C03641=1047.651,269.816,394.921,172.009,38.848,157.370
C03642=1047.658,270.065,394.890,172.012,38.851,157.371
C03643=1047.664,270.312,394.860,172.016,38.854,157.372
C03644=1047.670,270.561,394.829,172.018,38.856,157.372
C03645=1047.677,270.809,394.799,172.021,38.859,157.373
C03646=1047.683,271.057,394.769,172.023,38.862,157.374
C03647=1047.690,271.305,394.738,172.027,38.865,157.375
C03648=1047.697,271.553,394.708,172.030,38.868,157.375
C03649=1047.703,271.801,394.678,172.032,38.871,157.376
C03650=1047.710,272.049,394.648,172.036,38.874,157.377
C03651=1047.717,272.297,394.616,172.039,38.876,157.377
C03652=1047.723,272.545,394.586,172.041,38.879,157.378
C03653=1047.730,272.793,394.556,172.045,38.882,157.379
C03654=1047.736,273.041,394.525,172.047,38.885,157.379
C03655=1047.742,273.290,394.495,172.050,38.888,157.380
C03656=1047.749,273.537,394.464,172.054,38.891,157.381
C03657=1047.755,273.785,394.433,172.056,38.893,157.381
C03658=1047.762,274.034,394.403,172.059,38.896,157.382
C03659=1047.769,274.282,394.373,172.063,38.899,157.383
C03660=1047.775,274.529,394.342,172.065,38.902,157.384
C03661=1047.781,274.778,394.311,172.068,38.905,157.384
C03662=1047.789,275.026,394.281,172.072,38.908,157.385
C03663=1047.795,275.274,394.249,172.074,38.910,157.386
C03664=1047.801,275.521,394.219,172.077,38.913,157.386
C03665=1047.807,275.770,394.188,172.081,38.917,157.387
C03666=1047.815,276.018,394.157,172.083,38.919,157.388
C03667=1047.821,276.265,394.127,172.087,38.922,157.389
C03668=1047.828,276.535,394.093,172.089,38.925,157.389
C03669=1047.835,276.805,394.060,172.093,38.929,157.390
C03670=1047.842,277.075,394.026,172.096,38.931,157.391
C03671=1047.850,277.344,393.993,172.100,38.935,157.392
C03672=1047.856,277.592,393.962,172.102,38.938,157.392
C03673=1047.863,277.840,393.931,172.106,38.940,157.393
C03674=1047.869,278.089,393.900,172.109,38.943,157.394
C03675=1047.877,278.336,393.869,172.112,38.946,157.394
C03676=1047.882,278.584,393.839,172.115,38.949,157.395
C03677=1047.889,278.832,393.807,172.118,38.952,157.396
C03678=1047.895,279.081,393.777,172.121,38.955,157.397
C03679=1047.902,279.329,393.745,172.124,38.958,157.397
C03680=1047.908,279.576,393.714,172.128,38.961,157.398
C03681=1047.915,279.824,393.684,172.130,38.964,157.399
C03682=1047.921,280.072,393.652,172.133,38.966,157.399
C03683=1047.928,280.320,393.621,172.137,38.970,157.400
C03684=1047.935,280.569,393.590,172.139,38.973,157.401
C03685=1047.941,280.816,393.559,172.143,38.975,157.402
C03686=1047.947,281.064,393.527,172.145,38.978,157.402
C03687=1047.954,281.312,393.497,172.148,38.982,157.403
C03688=1047.961,281.560,393.465,172.152,38.984,157.404
C03689=1047.967,281.808,393.434,172.155,38.987,157.405
C03690=1047.973,282.055,393.403,172.158,38.990,157.405
C03691=1047.980,282.304,393.372,172.161,38.993,157.406
C03692=1047.987,282.552,393.341,172.165,38.996,157.407
C03693=1047.993,282.800,393.309,172.167,38.999,157.408
C03694=1048.000,283.048,393.278,172.171,39.002,157.408
C03695=1048.007,283.295,393.246,172.174,39.005,157.409
C03696=1048.013,283.544,393.216,172.177,39.008,157.410
C03697=1048.020,283.792,393.184,172.180,39.011,157.411
C03698=1048.026,284.039,393.153,172.184,39.014,157.411
C03699=1048.033,284.287,393.122,172.186,39.017,157.412
C03700=1048.040,284.535,393.090,172.189,39.020,157.413
C03701=1048.046,284.783,393.059,172.193,39.023,157.413
C03702=1048.053,285.031,393.027,172.195,39.026,157.414
C03703=1048.060,285.279,392.996,172.199,39.028,157.415
C03704=1048.066,285.526,392.965,172.202,39.032,157.416
C03705=1048.073,285.774,392.933,172.205,39.035,157.416
C03706=1048.080,286.022,392.902,172.209,39.037,157.417
C03707=1048.087,286.270,392.870,172.212,39.040,157.418
C03708=1048.093,286.518,392.839,172.216,39.044,157.419
C03709=1048.100,286.766,392.807,172.218,39.046,157.419
C03710=1048.106,287.014,392.775,172.222,39.049,157.420
C03711=1048.113,287.262,392.744,172.224,39.052,157.421
C03712=1048.119,287.510,392.713,172.228,39.055,157.422
C03713=1048.126,287.758,392.681,172.231,39.058,157.422
C03714=1048.133,288.006,392.650,172.235,39.061,157.423
C03715=1048.140,288.254,392.618,172.237,39.064,157.424
C03716=1048.146,288.502,392.586,172.241,39.067,157.425
C03717=1048.152,288.750,392.555,172.244,39.070,157.425
C03718=1048.159,288.997,392.523,172.247,39.073,157.426
C03719=1048.166,289.245,392.491,172.250,39.076,157.427
C03720=1048.172,289.493,392.459,172.254,39.079,157.428
C03721=1048.179,289.741,392.428,172.258,39.082,157.428
C03722=1048.186,289.989,392.396,172.260,39.085,157.429
C03723=1048.193,290.236,392.364,172.264,39.088,157.430
C03724=1048.200,290.518,392.328,172.268,39.092,157.431
C03725=1048.207,290.799,392.292,172.271,39.095,157.432
C03726=1048.215,291.080,392.255,172.274,39.099,157.433
C03727=1048.222,291.361,392.219,172.278,39.102,157.433
C03728=1048.229,291.610,392.187,172.282,39.105,157.434
C03729=1048.236,291.857,392.156,172.285,39.108,157.435
C03730=1048.242,292.105,392.123,172.288,39.111,157.436
C03731=1048.249,292.353,392.092,172.292,39.114,157.436
C03732=1048.255,292.601,392.060,172.295,39.118,157.437
C03733=1048.262,292.848,392.027,172.298,39.120,157.438
C03734=1048.268,293.096,391.996,172.301,39.123,157.439
C03735=1048.275,293.344,391.964,172.305,39.127,157.440
C03736=1048.281,293.592,391.932,172.309,39.129,157.440
C03737=1048.288,293.839,391.900,172.311,39.133,157.441
C03738=1048.295,294.088,391.867,172.315,39.135,157.442
C03739=1048.302,294.335,391.835,172.319,39.139,157.443
C03740=1048.308,294.584,391.803,172.321,39.142,157.443
C03741=1048.315,294.831,391.771,172.325,39.145,157.444
C03742=1048.322,295.079,391.740,172.328,39.148,157.445
C03743=1048.328,295.326,391.707,172.332,39.151,157.446
C03744=1048.335,295.574,391.675,172.335,39.154,157.447
C03745=1048.342,295.823,391.642,172.338,39.157,157.447
C03746=1048.349,296.070,391.610,172.342,39.160,157.448
C03747=1048.355,296.317,391.577,172.346,39.163,157.449
C03748=1048.361,296.566,391.545,172.348,39.167,157.450
C03749=1048.367,296.813,391.513,172.352,39.170,157.450
C03750=1048.374,297.061,391.480,172.356,39.173,157.451
C03751=1048.381,297.308,391.448,172.359,39.176,157.452
C03752=1048.387,297.557,391.415,172.363,39.180,157.453
C03753=1048.393,297.805,391.383,172.365,39.182,157.454
C03754=1048.400,298.052,391.350,172.369,39.186,157.455
C03755=1048.406,298.300,391.317,172.373,39.189,157.455
C03756=1048.413,298.547,391.285,172.375,39.192,157.456
C03757=1048.419,298.795,391.252,172.379,39.195,157.457
C03758=1048.426,299.043,391.219,172.383,39.199,157.458
C03759=1048.432,299.291,391.187,172.386,39.202,157.459
C03760=1048.439,299.538,391.155,172.390,39.205,157.459
C03761=1048.446,299.786,391.122,172.393,39.208,157.460
C03762=1048.452,300.034,391.089,172.396,39.211,157.461
C03763=1048.459,300.282,391.056,172.400,39.214,157.462
C03764=1048.465,300.529,391.024,172.404,39.217,157.463
C03765=1048.471,300.777,390.991,172.407,39.221,157.464
C03766=1048.479,301.025,390.958,172.410,39.224,157.464
C03767=1048.485,301.273,390.926,172.414,39.227,157.465
C03768=1048.492,301.520,390.893,172.418,39.230,157.466
C03769=1048.498,301.768,390.860,172.421,39.234,157.467
C03770=1048.505,302.016,390.827,172.424,39.237,157.468
C03771=1048.511,302.264,390.794,172.428,39.240,157.469
C03772=1048.518,302.511,390.762,172.432,39.243,157.469
C03773=1048.525,302.759,390.728,172.435,39.246,157.470
C03774=1048.532,303.006,390.696,172.438,39.250,157.471
C03775=1048.538,303.254,390.663,172.442,39.253,157.472
C03776=1048.545,303.502,390.630,172.446,39.256,157.473
C03777=1048.551,303.750,390.597,172.449,39.259,157.473
C03778=1048.558,303.997,390.565,172.453,39.263,157.474
C03779=1048.565,304.245,390.531,172.456,39.266,157.475
C03780=1048.573,304.542,390.491,172.460,39.270,157.476
C03781=1048.581,304.840,390.452,172.465,39.274,157.477
C03782=1048.589,305.137,390.412,172.469,39.278,157.478
C03783=1048.597,305.435,390.373,172.473,39.281,157.479
C03784=1048.604,305.682,390.340,172.477,39.285,157.480
C03785=1048.611,305.930,390.307,172.481,39.288,157.481
C03786=1048.617,306.178,390.274,172.484,39.291,157.482
C03787=1048.624,306.425,390.240,172.487,39.294,157.482
C03788=1048.630,306.673,390.207,172.491,39.297,157.483
C03789=1048.638,306.920,390.175,172.495,39.301,157.484
C03790=1048.645,307.168,390.141,172.499,39.304,157.485
C03791=1048.651,307.415,390.109,172.503,39.307,157.486
C03792=1048.658,307.664,390.075,172.506,39.311,157.487
C03793=1048.665,307.911,390.042,172.509,39.314,157.487
C03794=1048.671,308.159,390.009,172.513,39.317,157.488
C03795=1048.679,308.407,389.975,172.517,39.320,157.489
C03796=1048.685,308.654,389.942,172.521,39.323,157.490
C03797=1048.692,308.902,389.909,172.524,39.327,157.491
C03798=1048.699,309.149,389.876,172.528,39.330,157.492
C03799=1048.706,309.397,389.843,172.532,39.333,157.493
C03800=1048.713,309.644,389.810,172.535,39.337,157.493
C03801=1048.720,309.892,389.776,172.539,39.340,157.494
C03802=1048.726,310.140,389.743,172.542,39.343,157.495
C03803=1048.733,310.387,389.709,172.546,39.347,157.496
C03804=1048.740,310.636,389.676,172.550,39.350,157.497
C03805=1048.747,310.883,389.643,172.554,39.353,157.498
C03806=1048.754,311.130,389.609,172.558,39.356,157.498
C03807=1048.761,311.379,389.576,172.561,39.359,157.499
C03808=1048.768,311.626,389.542,172.565,39.363,157.500
C03809=1048.775,311.873,389.509,172.568,39.366,157.501
C03810=1048.782,312.122,389.476,172.572,39.369,157.502
C03811=1048.788,312.369,389.442,172.576,39.373,157.503
C03812=1048.796,312.616,389.409,172.580,39.376,157.504
C03813=1048.803,312.864,389.376,172.583,39.379,157.505
C03814=1048.809,313.111,389.342,172.587,39.383,157.506
C03815=1048.816,313.359,389.308,172.591,39.386,157.506
C03816=1048.822,313.606,389.274,172.595,39.390,157.507
C03817=1048.829,313.854,389.240,172.599,39.393,157.508
C03818=1048.836,314.102,389.206,172.603,39.397,157.509
C03819=1048.842,314.349,389.172,172.606,39.400,157.510
C03820=1048.849,314.597,389.138,172.610,39.403,157.511
C03821=1048.855,314.844,389.104,172.613,39.407,157.512
C03822=1048.862,315.092,389.070,172.617,39.411,157.513
C03823=1048.869,315.340,389.036,172.621,39.414,157.514
C03824=1048.875,315.587,389.002,172.625,39.417,157.514
C03825=1048.882,315.835,388.968,172.629,39.421,157.515
C03826=1048.888,316.083,388.934,172.633,39.424,157.516
C03827=1048.895,316.330,388.900,172.637,39.428,157.517
C03828=1048.902,316.578,388.866,172.641,39.432,157.518
C03829=1048.909,316.825,388.832,172.644,39.435,157.519
C03830=1048.915,317.073,388.798,172.648,39.438,157.520
C03831=1048.922,317.320,388.763,172.652,39.442,157.521
C03832=1048.929,317.568,388.729,172.655,39.445,157.522
C03833=1048.936,317.815,388.695,172.659,39.449,157.523
C03834=1048.942,318.063,388.661,172.663,39.452,157.524
C03835=1048.949,318.310,388.627,172.667,39.456,157.525
C03836=1048.957,318.612,388.586,172.672,39.460,157.526
C03837=1048.966,318.914,388.544,172.677,39.465,157.527
C03838=1048.974,319.216,388.502,172.681,39.469,157.528
C03839=1048.982,319.518,388.460,172.686,39.473,157.529
C03840=1048.989,319.765,388.425,172.690,39.477,157.530
C03841=1048.995,320.013,388.391,172.694,39.480,157.531
C03842=1049.002,320.260,388.357,172.698,39.484,157.532
C03843=1049.009,320.508,388.322,172.702,39.487,157.533
C03844=1049.016,320.755,388.288,172.706,39.491,157.534
C03845=1049.023,321.003,388.254,172.710,39.494,157.535
C03846=1049.030,321.250,388.219,172.714,39.498,157.536
C03847=1049.037,321.498,388.185,172.717,39.501,157.537
C03848=1049.043,321.746,388.150,172.721,39.505,157.538
C03849=1049.051,321.993,388.116,172.725,39.508,157.538
C03850=1049.056,322.241,388.082,172.729,39.512,157.539
C03851=1049.064,322.488,388.047,172.733,39.516,157.540
C03852=1049.070,322.736,388.013,172.737,39.519,157.541
C03853=1049.078,322.983,387.978,172.741,39.523,157.542
C03854=1049.084,323.231,387.944,172.745,39.527,157.543
C03855=1049.091,323.478,387.909,172.750,39.530,157.544
C03856=1049.099,323.725,387.874,172.754,39.534,157.545
C03857=1049.105,323.973,387.840,172.758,39.537,157.546
C03858=1049.113,324.220,387.805,172.762,39.541,157.547
C03859=1049.119,324.468,387.771,172.766,39.545,157.548
C03860=1049.126,324.716,387.736,172.769,39.548,157.549
C03861=1049.133,324.963,387.701,172.773,39.552,157.550
C03862=1049.140,325.211,387.667,172.777,39.555,157.551
C03863=1049.148,325.458,387.632,172.781,39.559,157.552
C03864=1049.155,325.706,387.597,172.785,39.563,157.553
C03865=1049.161,325.954,387.562,172.790,39.566,157.554
C03866=1049.169,326.201,387.528,172.794,39.570,157.555
C03867=1049.175,326.448,387.493,172.798,39.573,157.556
C03868=1049.183,326.695,387.458,172.802,39.577,157.557
C03869=1049.189,326.943,387.424,172.806,39.581,157.558
C03870=1049.196,327.191,387.388,172.810,39.584,157.559
C03871=1049.204,327.438,387.354,172.814,39.588,157.560
C03872=1049.211,327.686,387.318,172.819,39.591,157.561
C03873=1049.218,327.933,387.283,172.823,39.595,157.562
C03874=1049.225,328.181,387.249,172.827,39.599,157.563
C03875=1049.232,328.428,387.214,172.831,39.602,157.564
C03876=1049.238,328.675,387.179,172.835,39.606,157.565
C03877=1049.247,328.923,387.144,172.839,39.610,157.566
C03878=1049.253,329.171,387.109,172.844,39.613,157.566
C03879=1049.260,329.418,387.074,172.848,39.617,157.567
C03880=1049.268,329.665,387.039,172.852,39.621,157.568
C03881=1049.274,329.912,387.004,172.856,39.625,157.570
C03882=1049.282,330.160,386.969,172.860,39.629,157.571
C03883=1049.289,330.408,386.934,172.865,39.632,157.572
C03884=1049.295,330.655,386.899,172.869,39.636,157.573
C03885=1049.302,330.902,386.863,172.873,39.640,157.574
C03886=1049.309,331.149,386.828,172.877,39.644,157.575
C03887=1049.317,331.397,386.792,172.881,39.648,157.576
C03888=1049.323,331.645,386.757,172.886,39.651,157.577
C03889=1049.329,331.892,386.721,172.890,39.655,157.578
C03890=1049.336,332.139,386.685,172.894,39.659,157.579
C03891=1049.343,332.386,386.650,172.898,39.663,157.580
C03892=1049.352,332.683,386.608,172.903,39.667,157.581
C03893=1049.360,332.980,386.566,172.908,39.672,157.582
C03894=1049.369,333.277,386.523,172.913,39.676,157.583
C03895=1049.377,333.574,386.480,172.919,39.681,157.585
C03896=1049.384,333.821,386.445,172.923,39.685,157.586
C03897=1049.392,334.069,386.409,172.927,39.689,157.587
C03898=1049.398,334.316,386.374,172.931,39.693,157.588
C03899=1049.405,334.563,386.338,172.936,39.696,157.589
C03900=1049.413,334.811,386.302,172.940,39.700,157.590
C03901=1049.420,335.058,386.266,172.944,39.705,157.591
C03902=1049.427,335.305,386.231,172.949,39.708,157.592
C03903=1049.433,335.553,386.195,172.953,39.712,157.593
C03904=1049.440,335.800,386.159,172.957,39.716,157.594
C03905=1049.448,336.048,386.124,172.961,39.720,157.595
C03906=1049.455,336.295,386.088,172.966,39.724,157.596
C03907=1049.462,336.542,386.052,172.970,39.728,157.597
C03908=1049.469,336.790,386.016,172.974,39.732,157.598
C03909=1049.476,337.037,385.980,172.979,39.736,157.600
C03910=1049.483,337.284,385.944,172.983,39.740,157.601
C03911=1049.489,337.532,385.908,172.987,39.744,157.602
C03912=1049.496,337.779,385.872,172.993,39.748,157.603
C03913=1049.504,338.026,385.836,172.997,39.752,157.604
C03914=1049.510,338.273,385.800,173.001,39.756,157.605
C03915=1049.518,338.521,385.764,173.006,39.760,157.606
C03916=1049.525,338.768,385.728,173.010,39.764,157.607
C03917=1049.533,339.016,385.692,173.014,39.768,157.608
C03918=1049.539,339.263,385.656,173.019,39.772,157.609
C03919=1049.547,339.510,385.620,173.023,39.776,157.610
C03920=1049.553,339.757,385.584,173.027,39.780,157.611
C03921=1049.560,340.005,385.548,173.032,39.784,157.613
C03922=1049.567,340.252,385.512,173.037,39.788,157.614
C03923=1049.574,340.500,385.475,173.041,39.792,157.615
C03924=1049.581,340.746,385.439,173.046,39.796,157.616
C03925=1049.589,340.994,385.403,173.050,39.801,157.617
C03926=1049.595,341.241,385.366,173.055,39.804,157.618
C03927=1049.603,341.488,385.330,173.059,39.809,157.619
C03928=1049.611,341.736,385.294,173.063,39.812,157.620
C03929=1049.617,341.983,385.258,173.068,39.817,157.622
C03930=1049.625,342.230,385.221,173.073,39.821,157.623
C03931=1049.632,342.477,385.185,173.078,39.825,157.624
C03932=1049.639,342.725,385.149,173.082,39.829,157.625
C03933=1049.646,342.973,385.112,173.086,39.833,157.626
C03934=1049.653,343.219,385.076,173.091,39.837,157.627
C03935=1049.660,343.466,385.038,173.095,39.842,157.628
C03936=1049.667,343.713,385.003,173.100,39.846,157.630
C03937=1049.674,343.961,384.966,173.105,39.850,157.631
C03938=1049.682,344.208,384.930,173.110,39.854,157.632
C03939=1049.688,344.455,384.892,173.114,39.858,157.633
C03940=1049.695,344.703,384.856,173.119,39.863,157.634
C03941=1049.703,344.950,384.819,173.123,39.867,157.635
C03942=1049.710,345.196,384.782,173.127,39.871,157.636
C03943=1049.717,345.444,384.746,173.133,39.876,157.638
C03944=1049.724,345.692,384.709,173.137,39.879,157.639
C03945=1049.731,345.939,384.672,173.142,39.884,157.640
C03946=1049.738,346.185,384.636,173.146,39.888,157.641
C03947=1049.746,346.433,384.598,173.151,39.892,157.642
C03948=1049.755,346.726,384.555,173.157,39.898,157.644
C03949=1049.763,347.018,384.511,173.162,39.902,157.645
C03950=1049.771,347.312,384.467,173.167,39.907,157.646
C03951=1049.779,347.604,384.424,173.173,39.913,157.648
C03952=1049.787,347.851,384.387,173.178,39.917,157.649
C03953=1049.794,348.099,384.350,173.183,39.921,157.650
C03954=1049.801,348.346,384.312,173.188,39.926,157.651
C03955=1049.809,348.593,384.275,173.193,39.930,157.653
C03956=1049.816,348.840,384.239,173.197,39.934,157.654
C03957=1049.823,349.087,384.202,173.202,39.938,157.655
C03958=1049.830,349.334,384.164,173.206,39.943,157.656
C03959=1049.838,349.582,384.128,173.212,39.947,157.657
C03960=1049.845,349.829,384.090,173.216,39.952,157.659
C03961=1049.852,350.076,384.053,173.221,39.956,157.660
C03962=1049.859,350.324,384.016,173.226,39.960,157.661
C03963=1049.867,350.570,383.979,173.231,39.965,157.662
C03964=1049.874,350.817,383.942,173.236,39.969,157.664
C03965=1049.881,351.064,383.904,173.240,39.974,157.665
C03966=1049.888,351.311,383.867,173.245,39.978,157.666
C03967=1049.896,351.558,383.829,173.250,39.983,157.667
C03968=1049.903,351.805,383.792,173.255,39.987,157.669
C03969=1049.910,352.053,383.754,173.260,39.992,157.670
C03970=1049.917,352.300,383.717,173.265,39.996,157.671
C03971=1049.925,352.547,383.679,173.270,40.001,157.672
C03972=1049.932,352.794,383.642,173.275,40.005,157.673
C03973=1049.939,353.041,383.604,173.279,40.010,157.675
C03974=1049.946,353.288,383.567,173.285,40.014,157.676
C03975=1049.954,353.535,383.529,173.289,40.018,157.677
C03976=1049.961,353.782,383.492,173.294,40.023,157.679
C03977=1049.968,354.030,383.454,173.300,40.027,157.680
C03978=1049.975,354.277,383.416,173.304,40.032,157.681
C03979=1049.983,354.523,383.378,173.309,40.037,157.682
C03980=1049.990,354.770,383.341,173.315,40.041,157.684
C03981=1049.997,355.018,383.303,173.319,40.046,157.685
C03982=1050.005,355.265,383.266,173.324,40.051,157.686
C03983=1050.012,355.511,383.227,173.330,40.055,157.688
C03984=1050.019,355.758,383.190,173.334,40.060,157.689
C03985=1050.027,356.005,383.152,173.339,40.064,157.690
C03986=1050.034,356.253,383.115,173.344,40.069,157.691
C03987=1050.042,356.500,383.076,173.350,40.073,157.693
C03988=1050.049,356.747,383.039,173.354,40.078,157.694
C03989=1050.057,356.993,383.000,173.359,40.083,157.695
C03990=1050.064,357.241,382.963,173.365,40.087,157.697
C03991=1050.071,357.488,382.925,173.370,40.092,157.698
C03992=1050.079,357.734,382.887,173.375,40.097,157.699
C03993=1050.087,357.981,382.849,173.380,40.102,157.701
C03994=1050.094,358.229,382.810,173.385,40.106,157.702
C03995=1050.101,358.475,382.772,173.390,40.111,157.703
C03996=1050.108,358.723,382.735,173.395,40.116,157.704
C03997=1050.116,358.969,382.696,173.400,40.120,157.706
C03998=1050.123,359.216,382.659,173.406,40.125,157.707
C03999=1050.131,359.464,382.620,173.411,40.130,157.709
C04000=1050.138,359.710,382.581,173.416,40.135,157.710
C04001=1050.146,359.957,382.543,173.421,40.140,157.711
C04002=1050.153,360.204,382.506,173.426,40.144,157.713
C04003=1050.161,360.451,382.467,173.432,40.149,157.714
C04004=1050.170,360.749,382.421,173.438,40.155,157.716
C04005=1050.179,361.047,382.374,173.444,40.160,157.717
C04006=1050.188,361.346,382.328,173.451,40.166,157.719
C04007=1050.196,361.644,382.282,173.457,40.172,157.720
C04008=1050.204,361.891,382.243,173.462,40.177,157.722
C04009=1050.212,362.138,382.205,173.468,40.182,157.723
C04010=1050.219,362.384,382.167,173.473,40.187,157.725
C04011=1050.227,362.632,382.127,173.478,40.192,157.726
C04012=1050.234,362.878,382.089,173.483,40.197,157.727
C04013=1050.242,363.125,382.051,173.488,40.201,157.729
C04014=1050.249,363.372,382.012,173.494,40.207,157.730
C04015=1050.257,363.619,381.973,173.499,40.211,157.732
C04016=1050.264,363.866,381.934,173.505,40.217,157.733
C04017=1050.272,364.112,381.895,173.510,40.222,157.734
C04018=1050.279,364.359,381.856,173.516,40.226,157.736
C04019=1050.286,364.607,381.817,173.521,40.232,157.737
C04020=1050.294,364.853,381.779,173.526,40.236,157.739
C04021=1050.301,365.101,381.740,173.531,40.242,157.740
C04022=1050.309,365.346,381.701,173.537,40.247,157.742
C04023=1050.316,365.593,381.662,173.542,40.252,157.743
C04024=1050.324,365.840,381.623,173.548,40.257,157.744
C04025=1050.331,366.087,381.584,173.553,40.262,157.746
C04026=1050.339,366.334,381.545,173.559,40.267,157.747
C04027=1050.346,366.581,381.506,173.564,40.272,157.749
C04028=1050.354,366.828,381.466,173.570,40.277,157.750
C04029=1050.362,367.074,381.428,173.575,40.282,157.752
C04030=1050.369,367.321,381.388,173.581,40.287,157.753
C04031=1050.377,367.568,381.350,173.586,40.292,157.755
C04032=1050.384,367.814,381.310,173.592,40.297,157.756
C04033=1050.393,368.062,381.271,173.597,40.303,157.758
C04034=1050.400,368.308,381.232,173.603,40.308,157.759
C04035=1050.407,368.555,381.193,173.609,40.313,157.760
C04036=1050.415,368.801,381.154,173.614,40.318,157.762
C04037=1050.423,369.048,381.114,173.620,40.323,157.764
C04038=1050.431,369.295,381.075,173.625,40.329,157.765
C04039=1050.438,369.542,381.036,173.631,40.334,157.767
C04040=1050.446,369.789,380.996,173.636,40.339,157.768
C04041=1050.454,370.036,380.957,173.642,40.344,157.769
C04042=1050.461,370.282,380.918,173.648,40.349,157.771
C04043=1050.469,370.529,380.878,173.653,40.354,157.772
C04044=1050.477,370.775,380.838,173.659,40.360,157.774
C04045=1050.485,371.023,380.799,173.664,40.365,157.776
C04046=1050.492,371.269,380.760,173.670,40.370,157.777
C04047=1050.500,371.516,380.720,173.676,40.376,157.779
C04048=1050.508,371.763,380.680,173.681,40.381,157.780
C04049=1050.516,372.010,380.640,173.688,40.386,157.782
C04050=1050.523,372.256,380.601,173.694,40.392,157.783
C04051=1050.530,372.503,380.561,173.699,40.397,157.785
C04052=1050.538,372.750,380.521,173.705,40.402,157.786
C04053=1050.547,372.996,380.482,173.711,40.408,157.788
C04054=1050.554,373.242,380.442,173.716,40.414,157.790
C04055=1050.562,373.489,380.402,173.722,40.419,157.791
C04056=1050.569,373.736,380.362,173.728,40.424,157.793
C04057=1050.577,373.983,380.322,173.733,40.430,157.794
C04058=1050.585,374.229,380.282,173.740,40.435,157.796
C04059=1050.592,374.476,380.242,173.746,40.440,157.797
C04060=1050.603,374.793,380.191,173.753,40.448,157.799
C04061=1050.612,375.110,380.139,173.760,40.455,157.801
C04062=1050.623,375.428,380.087,173.768,40.462,157.804
C04063=1050.632,375.745,380.035,173.775,40.469,157.806
C04064=1050.640,375.991,379.996,173.781,40.475,157.807
C04065=1050.648,376.238,379.955,173.788,40.480,157.809
C04066=1050.656,376.485,379.915,173.794,40.486,157.810
C04067=1050.664,376.731,379.874,173.799,40.491,157.812
C04068=1050.671,376.978,379.834,173.805,40.497,157.814
C04069=1050.679,377.224,379.794,173.811,40.503,157.815
C04070=1050.687,377.471,379.754,173.818,40.508,157.817
C04071=1050.695,377.717,379.713,173.823,40.513,157.819
C04072=1050.704,377.964,379.674,173.829,40.519,157.820
C04073=1050.712,378.210,379.633,173.836,40.525,157.822
C04074=1050.720,378.456,379.593,173.842,40.531,157.824
C04075=1050.727,378.703,379.553,173.848,40.537,157.825
C04076=1050.735,378.950,379.512,173.853,40.542,157.827
C04077=1050.743,379.196,379.471,173.860,40.548,157.829
C04078=1050.752,379.443,379.430,173.866,40.553,157.830
C04079=1050.760,379.690,379.391,173.872,40.559,157.832
C04080=1050.767,379.936,379.349,173.879,40.565,157.834
C04081=1050.775,380.183,379.309,173.884,40.571,157.835
C04082=1050.783,380.429,379.268,173.890,40.576,157.837
C04083=1050.790,380.676,379.227,173.897,40.582,157.839
C04084=1050.798,380.922,379.186,173.903,40.588,157.841
C04085=1050.806,381.168,379.146,173.909,40.594,157.842
C04086=1050.814,381.414,379.105,173.916,40.600,157.844
C04087=1050.822,381.662,379.063,173.922,40.606,157.846
C04088=1050.830,381.908,379.023,173.928,40.612,157.848
C04089=1050.838,382.154,378.982,173.934,40.618,157.849
C04090=1050.846,382.400,378.940,173.940,40.624,157.851
C04091=1050.854,382.647,378.899,173.946,40.630,157.853
C04092=1050.863,382.894,378.858,173.953,40.636,157.854
C04093=1050.870,383.140,378.817,173.959,40.642,157.856
C04094=1050.878,383.386,378.777,173.966,40.648,157.858
C04095=1050.886,383.632,378.735,173.972,40.653,157.860
C04096=1050.894,383.879,378.694,173.979,40.660,157.862
C04097=1050.902,384.126,378.653,173.985,40.665,157.863
C04098=1050.911,384.371,378.612,173.991,40.672,157.865
C04099=1050.918,384.619,378.570,173.998,40.678,157.867
C04100=1050.927,384.864,378.529,174.004,40.684,157.869
C04101=1050.935,385.111,378.488,174.011,40.690,157.871
C04102=1050.943,385.357,378.446,174.017,40.696,157.872
C04103=1050.951,385.604,378.405,174.023,40.702,157.874
C04104=1050.959,385.850,378.363,174.030,40.708,157.876
C04105=1050.967,386.096,378.322,174.037,40.714,157.878
C04106=1050.976,386.342,378.281,174.043,40.721,157.880
C04107=1050.983,386.589,378.239,174.049,40.726,157.881
C04108=1050.992,386.835,378.198,174.055,40.733,157.883
C04109=1051.001,387.081,378.156,174.063,40.739,157.885
C04110=1051.008,387.328,378.115,174.070,40.745,157.887
C04111=1051.017,387.574,378.073,174.076,40.751,157.889
C04112=1051.025,387.820,378.031,174.083,40.757,157.891
C04113=1051.033,388.067,377.990,174.089,40.764,157.893
C04114=1051.042,388.313,377.948,174.096,40.770,157.894
C04115=1051.050,388.560,377.907,174.103,40.776,157.896
C04116=1051.062,388.909,377.847,174.112,40.785,157.899
C04117=1051.074,389.259,377.787,174.122,40.794,157.902
C04118=1051.085,389.609,377.729,174.131,40.803,157.904
C04119=1051.097,389.958,377.669,174.141,40.812,157.907
C04120=1051.105,390.205,377.627,174.147,40.819,157.909
C04121=1051.113,390.451,377.585,174.154,40.825,157.911
C04122=1051.122,390.697,377.542,174.161,40.832,157.913
C04123=1051.130,390.943,377.500,174.167,40.838,157.915
C04124=1051.138,391.189,377.458,174.174,40.844,157.917
C04125=1051.147,391.436,377.416,174.182,40.851,157.919
C04126=1051.155,391.682,377.373,174.189,40.858,157.921
C04127=1051.163,391.928,377.331,174.195,40.864,157.923
C04128=1051.172,392.174,377.290,174.202,40.870,157.925
C04129=1051.180,392.420,377.247,174.209,40.877,157.927
C04130=1051.189,392.667,377.204,174.215,40.883,157.929
C04131=1051.197,392.914,377.162,174.223,40.890,157.931
C04132=1051.205,393.159,377.120,174.230,40.897,157.933
C04133=1051.214,393.405,377.078,174.237,40.904,157.935
C04134=1051.222,393.651,377.035,174.243,40.910,157.937
C04135=1051.231,393.897,376.992,174.251,40.917,157.939
C04136=1051.239,394.144,376.949,174.258,40.923,157.941
C04137=1051.247,394.389,376.907,174.265,40.930,157.943
C04138=1051.256,394.636,376.865,174.272,40.937,157.945
C04139=1051.264,394.882,376.822,174.279,40.943,157.947
C04140=1051.273,395.128,376.779,174.286,40.950,157.949
C04141=1051.281,395.374,376.736,174.293,40.957,157.951
C04142=1051.289,395.621,376.693,174.301,40.964,157.953
C04143=1051.298,395.867,376.650,174.308,40.971,157.955
C04144=1051.306,396.113,376.607,174.315,40.977,157.957
C04145=1051.316,396.358,376.565,174.322,40.984,157.959
C04146=1051.324,396.605,376.522,174.330,40.991,157.961
C04147=1051.333,396.851,376.479,174.336,40.998,157.963
C04148=1051.341,397.097,376.436,174.343,41.005,157.965
C04149=1051.350,397.343,376.393,174.351,41.012,157.968
C04150=1051.357,397.589,376.349,174.358,41.019,157.970
C04151=1051.366,397.835,376.306,174.366,41.026,157.972
C04152=1051.374,398.081,376.263,174.373,41.032,157.974
C04153=1051.383,398.327,376.220,174.381,41.040,157.976
C04154=1051.392,398.573,376.176,174.388,41.047,157.978
C04155=1051.400,398.819,376.133,174.395,41.053,157.980
C04156=1051.409,399.065,376.090,174.403,41.061,157.983
C04157=1051.418,399.311,376.047,174.410,41.068,157.985
C04158=1051.427,399.557,376.003,174.418,41.075,157.987
C04159=1051.435,399.803,375.960,174.425,41.082,157.989
C04160=1051.444,400.049,375.917,174.433,41.089,157.991
C04161=1051.453,400.295,375.873,174.440,41.096,157.993
C04162=1051.461,400.541,375.830,174.448,41.103,157.996
C04163=1051.470,400.787,375.786,174.455,41.110,157.998
C04164=1051.478,401.033,375.743,174.463,41.118,158.000
C04165=1051.487,401.279,375.699,174.470,41.125,158.002
C04166=1051.496,401.525,375.656,174.478,41.132,158.005
C04167=1051.505,401.771,375.612,174.485,41.139,158.007
C04168=1051.513,402.018,375.568,174.493,41.147,158.009
C04169=1051.522,402.263,375.524,174.500,41.154,158.011
C04170=1051.531,402.509,375.480,174.509,41.161,158.014
C04171=1051.540,402.755,375.436,174.516,41.168,158.016
C04172=1051.547,402.968,375.398,174.523,41.175,158.018
C04173=1051.555,403.182,375.360,174.530,41.182,158.020
C04174=1051.562,403.395,375.322,174.536,41.188,158.022
C04175=1051.570,403.609,375.284,174.544,41.194,158.024
C04176=1051.584,404.009,375.212,174.556,41.206,158.028
C04177=1051.598,404.410,375.140,174.568,41.218,158.031
C04178=1051.613,404.810,375.068,174.581,41.231,158.035
C04179=1051.628,405.211,374.996,174.594,41.243,158.039
C04180=1051.636,405.457,374.951,174.602,41.250,158.041
C04181=1051.645,405.703,374.907,174.610,41.258,158.044
C04182=1051.654,405.949,374.862,174.618,41.266,158.046
C04183=1051.663,406.195,374.818,174.626,41.274,158.049
C04184=1051.671,406.440,374.773,174.634,41.281,158.051
C04185=1051.681,406.686,374.729,174.642,41.289,158.053
C04186=1051.690,406.933,374.684,174.650,41.296,158.056
C04187=1051.699,407.178,374.640,174.659,41.305,158.058
C04188=1051.707,407.424,374.595,174.667,41.312,158.061
C04189=1051.716,407.670,374.550,174.674,41.320,158.063
C04190=1051.725,407.915,374.506,174.683,41.327,158.066
C04191=1051.734,408.161,374.461,174.691,41.336,158.068
C04192=1051.743,408.407,374.417,174.699,41.343,158.070
C04193=1051.752,408.653,374.371,174.708,41.351,158.073
C04194=1051.762,408.899,374.326,174.716,41.359,158.075
C04195=1051.770,409.144,374.282,174.724,41.367,158.078
C04196=1051.779,409.390,374.237,174.732,41.375,158.080
C04197=1051.789,409.636,374.192,174.741,41.383,158.083
C04198=1051.798,409.882,374.146,174.749,41.390,158.085
C04199=1051.807,410.128,374.102,174.758,41.398,158.088
C04200=1051.816,410.374,374.057,174.766,41.407,158.091
C04201=1051.825,410.619,374.011,174.775,41.415,158.093
C04202=1051.835,410.865,373.967,174.783,41.423,158.096
C04203=1051.844,411.111,373.921,174.792,41.430,158.098
C04204=1051.853,411.357,373.876,174.800,41.438,158.101
C04205=1051.863,411.602,373.831,174.809,41.446,158.103
C04206=1051.872,411.848,373.785,174.817,41.455,158.106
C04207=1051.881,412.093,373.741,174.826,41.463,158.108
C04208=1051.890,412.339,373.695,174.835,41.471,158.111
C04209=1051.900,412.584,373.649,174.843,41.479,158.114
C04210=1051.909,412.830,373.604,174.852,41.487,158.116
C04211=1051.918,413.076,373.559,174.861,41.495,158.119
C04212=1051.928,413.322,373.513,174.869,41.504,158.122
C04213=1051.937,413.568,373.467,174.878,41.512,158.124
C04214=1051.946,413.813,373.422,174.887,41.521,158.127
C04215=1051.955,414.059,373.375,174.895,41.529,158.130
C04216=1051.964,414.304,373.330,174.904,41.537,158.132
C04217=1051.974,414.550,373.284,174.914,41.546,158.135
C04218=1051.983,414.796,373.238,174.923,41.554,158.138
C04219=1051.993,415.041,373.192,174.931,41.562,158.140
C04220=1052.002,415.286,373.146,174.940,41.571,158.143
C04221=1052.011,415.532,373.100,174.949,41.579,158.146
C04222=1052.021,415.778,373.054,174.959,41.588,158.149
C04223=1052.031,416.023,373.008,174.967,41.597,158.151
C04224=1052.040,416.268,372.962,174.976,41.605,158.154
C04225=1052.050,416.515,372.916,174.985,41.614,158.157
C04226=1052.059,416.760,372.870,174.994,41.622,158.160
C04227=1052.069,417.006,372.824,175.004,41.631,158.162
C04228=1052.083,417.380,372.753,175.018,41.644,158.167
C04229=1052.098,417.755,372.683,175.032,41.657,158.171
C04230=1052.112,418.129,372.612,175.046,41.671,158.175
C04231=1052.127,418.504,372.540,175.060,41.684,158.180
C04232=1052.136,418.749,372.494,175.069,41.693,158.183
C04233=1052.146,418.995,372.447,175.079,41.702,158.186
C04234=1052.156,419.241,372.401,175.088,41.710,158.188
C04235=1052.165,419.485,372.354,175.098,41.719,158.191
C04236=1052.175,419.731,372.307,175.107,41.728,158.194
C04237=1052.185,419.977,372.261,175.117,41.737,158.197
C04238=1052.194,420.222,372.213,175.126,41.746,158.200
C04239=1052.204,420.468,372.167,175.136,41.755,158.203
C04240=1052.213,420.713,372.120,175.146,41.764,158.206
C04241=1052.224,420.958,372.073,175.156,41.773,158.209
C04242=1052.233,421.204,372.026,175.165,41.782,158.212
C04243=1052.242,421.449,371.979,175.175,41.791,158.215
C04244=1052.253,421.694,371.932,175.184,41.800,158.218
C04245=1052.262,421.940,371.884,175.194,41.810,158.221
C04246=1052.272,422.186,371.837,175.205,41.819,158.224
C04247=1052.282,422.431,371.790,175.214,41.828,158.227
C04248=1052.291,422.676,371.743,175.224,41.837,158.230
C04249=1052.301,422.921,371.696,175.234,41.847,158.233
C04250=1052.311,423.166,371.648,175.244,41.856,158.236
C04251=1052.322,423.412,371.601,175.254,41.865,158.239
C04252=1052.331,423.657,371.553,175.264,41.874,158.242
C04253=1052.341,423.902,371.505,175.274,41.884,158.246
C04254=1052.352,424.147,371.458,175.284,41.893,158.249
C04255=1052.361,424.393,371.410,175.294,41.903,158.252
C04256=1052.371,424.638,371.363,175.304,41.912,158.255
C04257=1052.382,424.883,371.316,175.314,41.921,158.258
C04258=1052.391,425.128,371.267,175.325,41.931,158.261
C04259=1052.401,425.374,371.220,175.335,41.940,158.264
C04260=1052.411,425.618,371.172,175.345,41.950,158.268
C04261=1052.421,425.864,371.124,175.356,41.959,158.271
C04262=1052.431,426.109,371.076,175.365,41.969,158.274
C04263=1052.441,426.354,371.029,175.376,41.978,158.277
C04264=1052.452,426.600,370.980,175.386,41.988,158.281
C04265=1052.462,426.844,370.932,175.397,41.998,158.284
C04266=1052.472,427.090,370.884,175.408,42.007,158.287
C04267=1052.481,427.335,370.836,175.418,42.017,158.290
C04268=1052.492,427.580,370.788,175.429,42.027,158.294
C04269=1052.502,427.825,370.739,175.439,42.037,158.297
C04270=1052.513,428.070,370.691,175.450,42.047,158.300
C04271=1052.523,428.315,370.642,175.461,42.057,158.304
C04272=1052.534,428.560,370.594,175.471,42.067,158.307
C04273=1052.543,428.805,370.545,175.482,42.077,158.311
C04274=1052.553,429.050,370.497,175.493,42.087,158.314
C04275=1052.564,429.296,370.449,175.504,42.096,158.317
C04276=1052.574,429.541,370.400,175.515,42.107,158.321
C04277=1052.585,429.786,370.350,175.526,42.117,158.324
C04278=1052.595,430.030,370.303,175.537,42.127,158.328
C04279=1052.605,430.275,370.254,175.548,42.137,158.331
C04280=1052.616,430.520,370.204,175.559,42.147,158.334
C04281=1052.625,430.765,370.156,175.570,42.157,158.338
C04282=1052.636,431.010,370.106,175.581,42.167,158.341
C04283=1052.646,431.255,370.058,175.592,42.178,158.345
C04284=1052.663,431.652,369.978,175.610,42.194,158.351
C04285=1052.680,432.049,369.898,175.629,42.211,158.356
C04286=1052.697,432.446,369.818,175.647,42.228,158.362
C04287=1052.714,432.843,369.738,175.665,42.245,158.368
C04288=1052.725,433.088,369.689,175.677,42.255,158.372
C04289=1052.736,433.333,369.640,175.688,42.266,158.375
C04290=1052.746,433.577,369.591,175.701,42.277,158.379
C04291=1052.757,433.822,369.541,175.712,42.287,158.383
C04292=1052.768,434.067,369.491,175.724,42.297,158.386
C04293=1052.778,434.312,369.441,175.735,42.308,158.390
C04294=1052.789,434.557,369.391,175.747,42.319,158.394
C04295=1052.799,434.801,369.342,175.758,42.330,158.397
C04296=1052.810,435.046,369.292,175.771,42.340,158.401
C04297=1052.821,435.290,369.243,175.782,42.351,158.405
C04298=1052.832,435.535,369.193,175.794,42.362,158.409
C04299=1052.843,435.780,369.143,175.806,42.373,158.412
C04300=1052.854,436.025,369.093,175.818,42.383,158.416
C04301=1052.865,436.270,369.043,175.830,42.394,158.420
C04302=1052.876,436.515,368.993,175.843,42.405,158.424
C04303=1052.887,436.760,368.943,175.855,42.416,158.428
C04304=1052.898,437.004,368.892,175.866,42.427,158.431
C04305=1052.909,437.248,368.842,175.879,42.438,158.435
C04306=1052.920,437.493,368.792,175.891,42.449,158.439
C04307=1052.930,437.738,368.741,175.904,42.460,158.443
C04308=1052.941,437.983,368.691,175.916,42.471,158.447
C04309=1052.953,438.227,368.640,175.929,42.482,158.451
C04310=1052.964,438.472,368.589,175.940,42.493,158.455
C04311=1052.975,438.716,368.539,175.954,42.505,158.459
C04312=1052.986,438.960,368.489,175.965,42.516,158.463
C04313=1052.997,439.206,368.438,175.979,42.528,158.467
C04314=1053.008,439.450,368.386,175.991,42.538,158.471
C04315=1053.019,439.694,368.336,176.004,42.550,158.475
C04316=1053.030,439.939,368.285,176.017,42.562,158.479
C04317=1053.041,440.183,368.234,176.030,42.573,158.483
C04318=1053.052,440.428,368.183,176.043,42.584,158.487
C04319=1053.064,440.672,368.132,176.055,42.596,158.491
C04320=1053.075,440.916,368.081,176.068,42.607,158.496
C04321=1053.086,441.162,368.030,176.081,42.619,158.500
C04322=1053.097,441.405,367.979,176.095,42.631,158.504
C04323=1053.109,441.650,367.927,176.108,42.642,158.508
C04324=1053.121,441.894,367.876,176.121,42.654,158.512
C04325=1053.131,442.139,367.824,176.134,42.665,158.516
C04326=1053.143,442.383,367.773,176.148,42.677,158.521
C04327=1053.154,442.628,367.721,176.160,42.689,158.525
C04328=1053.166,442.872,367.670,176.174,42.701,158.529
C04329=1053.177,443.116,367.618,176.188,42.713,158.534
C04330=1053.189,443.361,367.566,176.201,42.725,158.538
C04331=1053.200,443.604,367.515,176.215,42.737,158.542
C04332=1053.211,443.849,367.463,176.228,42.749,158.547
C04333=1053.223,444.093,367.411,176.242,42.761,158.551
C04334=1053.235,444.337,367.359,176.255,42.773,158.555
C04335=1053.247,444.582,367.307,176.269,42.785,158.560
C04336=1053.259,444.826,367.255,176.284,42.797,158.564
C04337=1053.269,445.070,367.203,176.297,42.809,158.569
C04338=1053.281,445.314,367.151,176.311,42.821,158.573
C04339=1053.293,445.558,367.099,176.325,42.834,158.578
C04340=1053.305,445.784,367.051,176.338,42.845,158.582
C04341=1053.315,446.009,367.002,176.351,42.856,158.586
C04342=1053.326,446.234,366.954,176.364,42.868,158.590
C04343=1053.337,446.459,366.906,176.377,42.880,158.595
C04344=1053.349,446.685,366.858,176.390,42.891,158.599
C04345=1053.361,446.911,366.811,176.403,42.901,158.603
C04346=1053.374,447.138,366.763,176.418,42.912,158.607
C04347=1053.388,447.365,366.717,176.431,42.924,158.611
C04348=1053.404,447.609,366.667,176.445,42.935,158.615
C04349=1053.420,447.852,366.618,176.460,42.946,158.620
C04350=1053.436,448.097,366.570,176.474,42.958,158.624
C04351=1053.455,448.341,366.522,176.490,42.968,158.628
C04352=1053.473,448.586,366.474,176.504,42.979,158.632
C04353=1053.493,448.831,366.427,176.519,42.989,158.637
C04354=1053.512,449.076,366.382,176.534,43.000,158.641
C04355=1053.534,449.321,366.335,176.549,43.010,158.645
C04356=1053.555,449.566,366.291,176.565,43.021,158.649
C04357=1053.577,449.812,366.246,176.580,43.031,158.653
C04358=1053.600,450.056,366.203,176.595,43.040,158.657
C04359=1053.624,450.301,366.159,176.610,43.050,158.661
C04360=1053.305,450.324,365.866,176.609,43.149,158.689
C04361=1053.281,450.079,365.908,176.594,43.139,158.685
C04362=1053.258,449.833,365.953,176.578,43.129,158.681
C04363=1053.236,449.588,365.997,176.563,43.120,158.677
C04364=1053.213,449.343,366.043,176.548,43.110,158.673
C04365=1053.193,449.098,366.088,176.532,43.099,158.669
C04366=1053.172,448.852,366.134,176.517,43.089,158.665
C04367=1053.154,448.608,366.181,176.502,43.078,158.661
C04368=1053.134,448.364,366.228,176.488,43.068,158.656
C04369=1053.116,448.119,366.277,176.472,43.057,158.652
C04370=1053.099,447.874,366.324,176.458,43.045,158.648
C04371=1053.083,447.630,366.373,176.443,43.034,158.643
C04372=1053.067,447.387,366.422,176.429,43.023,158.639
C04373=1053.054,447.169,366.467,176.416,43.013,158.635
C04374=1053.041,446.952,366.512,176.403,43.002,158.631
C04375=1053.028,446.734,366.557,176.389,42.991,158.627
C04376=1053.017,446.519,366.603,176.377,42.981,158.623
C04377=1053.006,446.302,366.650,176.364,42.970,158.619
C04378=1052.996,446.087,366.696,176.351,42.959,158.615
C04379=1052.985,445.871,366.742,176.339,42.948,158.611
C04380=1052.974,445.655,366.788,176.326,42.938,158.607
C04381=1052.963,445.411,366.840,176.312,42.925,158.603
C04382=1052.951,445.167,366.892,176.299,42.914,158.598
C04383=1052.939,444.923,366.945,176.284,42.901,158.594
C04384=1052.927,444.679,366.997,176.270,42.889,158.589
C04385=1052.916,444.434,367.049,176.257,42.877,158.585
C04386=1052.904,444.190,367.101,176.243,42.865,158.580
C04387=1052.893,443.946,367.152,176.228,42.853,158.576
C04388=1052.881,443.702,367.205,176.215,42.841,158.572
C04389=1052.869,443.457,367.256,176.201,42.830,158.567
C04390=1052.858,443.213,367.308,176.188,42.818,158.563
C04391=1052.846,442.968,367.360,176.174,42.806,158.559
C04392=1052.835,442.725,367.412,176.161,42.794,158.554
C04393=1052.823,442.480,367.464,176.147,42.782,158.550
C04394=1052.812,442.236,367.515,176.134,42.770,158.546
C04395=1052.801,441.991,367.567,176.121,42.759,158.542
C04396=1052.789,441.747,367.618,176.107,42.747,158.537
C04397=1052.777,441.502,367.669,176.094,42.736,158.533
C04398=1052.766,441.258,367.720,176.081,42.724,158.529
C04399=1052.755,441.013,367.772,176.068,42.712,158.525
C04400=1052.744,440.769,367.823,176.054,42.701,158.521
C04401=1052.732,440.525,367.874,176.041,42.690,158.516
C04402=1052.721,440.280,367.924,176.029,42.678,158.512
C04403=1052.710,440.036,367.976,176.016,42.667,158.508
C04404=1052.699,439.791,368.027,176.003,42.655,158.504
C04405=1052.688,439.547,368.078,175.990,42.644,158.500
C04406=1052.676,439.302,368.129,175.978,42.633,158.496
C04407=1052.666,439.058,368.180,175.965,42.622,158.492
C04408=1052.655,438.814,368.230,175.951,42.610,158.488
C04409=1052.643,438.569,368.281,175.940,42.599,158.484
C04410=1052.632,438.324,368.331,175.927,42.588,158.480
C04411=1052.621,438.080,368.382,175.915,42.576,158.476
C04412=1052.610,437.835,368.432,175.902,42.566,158.472
C04413=1052.598,437.590,368.483,175.890,42.554,158.468
C04414=1052.588,437.345,368.534,175.877,42.543,158.464
C04415=1052.577,437.101,368.584,175.865,42.532,158.460
C04416=1052.566,436.857,368.634,175.852,42.522,158.457
C04417=1052.555,436.612,368.685,175.840,42.511,158.453
C04418=1052.545,436.367,368.734,175.828,42.500,158.449
C04419=1052.534,436.123,368.785,175.816,42.489,158.445
C04420=1052.522,435.877,368.835,175.804,42.478,158.441
C04421=1052.511,435.632,368.885,175.791,42.467,158.437
C04422=1052.500,435.388,368.935,175.780,42.457,158.434
C04423=1052.489,435.143,368.984,175.768,42.446,158.430
C04424=1052.478,434.898,369.034,175.756,42.436,158.426
C04425=1052.467,434.654,369.084,175.744,42.425,158.422
C04426=1052.457,434.409,369.133,175.732,42.414,158.419
C04427=1052.447,434.164,369.183,175.721,42.404,158.415
C04428=1052.436,433.920,369.233,175.708,42.393,158.411
C04429=1052.425,433.675,369.283,175.697,42.383,158.408
C04430=1052.414,433.430,369.333,175.685,42.372,158.404
C04431=1052.403,433.185,369.382,175.674,42.361,158.400
C04432=1052.393,432.941,369.431,175.662,42.351,158.397
C04433=1052.376,432.541,369.511,175.643,42.334,158.391
C04434=1052.358,432.143,369.592,175.625,42.317,158.385
C04435=1052.342,431.743,369.673,175.607,42.301,158.379
C04436=1052.325,431.344,369.752,175.588,42.284,158.373
C04437=1052.313,431.099,369.801,175.576,42.274,158.370
C04438=1052.304,430.854,369.850,175.565,42.264,158.366
C04439=1052.293,430.609,369.899,175.555,42.253,158.363
C04440=1052.283,430.365,369.949,175.543,42.243,158.359
C04441=1052.273,430.119,369.998,175.532,42.233,158.356
C04442=1052.263,429.874,370.046,175.521,42.223,158.352
C04443=1052.251,429.630,370.095,175.510,42.213,158.349
C04444=1052.242,429.385,370.144,175.499,42.203,158.346
C04445=1052.231,429.139,370.192,175.488,42.193,158.342
C04446=1052.221,428.894,370.240,175.477,42.184,158.339
C04447=1052.211,428.649,370.289,175.466,42.173,158.335
C04448=1052.200,428.405,370.338,175.455,42.163,158.332
C04449=1052.190,428.160,370.386,175.445,42.154,158.329
C04450=1052.180,427.915,370.435,175.434,42.144,158.325
C04451=1052.169,427.669,370.483,175.423,42.134,158.322
C04452=1052.160,427.424,370.531,175.413,42.124,158.319
C04453=1052.149,427.179,370.579,175.402,42.115,158.315
C04454=1052.139,426.934,370.628,175.391,42.105,158.312
C04455=1052.128,426.689,370.676,175.381,42.095,158.309
C04456=1052.118,426.444,370.724,175.370,42.086,158.306
C04457=1052.109,426.198,370.772,175.360,42.076,158.302
C04458=1052.099,425.954,370.820,175.349,42.067,158.299
C04459=1052.089,425.708,370.868,175.339,42.057,158.296
C04460=1052.079,425.463,370.916,175.328,42.048,158.293
C04461=1052.068,425.218,370.963,175.318,42.038,158.289
C04462=1052.059,424.973,371.012,175.308,42.029,158.286
C04463=1052.048,424.727,371.059,175.298,42.019,158.283
C04464=1052.038,424.482,371.106,175.287,42.010,158.280
C04465=1052.028,424.237,371.155,175.277,42.001,158.277
C04466=1052.018,423.991,371.202,175.268,41.991,158.274
C04467=1052.008,423.746,371.249,175.257,41.982,158.271
C04468=1051.998,423.501,371.297,175.247,41.972,158.267
C04469=1051.988,423.255,371.344,175.237,41.963,158.264
C04470=1051.978,423.011,371.391,175.227,41.954,158.261
C04471=1051.969,422.765,371.439,175.217,41.945,158.258
C04472=1051.959,422.520,371.486,175.207,41.936,158.255
C04473=1051.948,422.275,371.534,175.196,41.926,158.252
C04474=1051.939,422.029,371.581,175.187,41.918,158.249
C04475=1051.929,421.784,371.629,175.177,41.908,158.246
C04476=1051.919,421.539,371.675,175.168,41.899,158.243
C04477=1051.909,421.294,371.723,175.158,41.890,158.240
C04478=1051.900,421.048,371.770,175.148,41.881,158.237
C04479=1051.890,420.802,371.817,175.138,41.872,158.234
C04480=1051.880,420.558,371.864,175.128,41.863,158.231
C04481=1051.871,420.312,371.911,175.119,41.854,158.228
C04482=1051.861,420.066,371.958,175.109,41.845,158.225
C04483=1051.851,419.821,372.004,175.100,41.836,158.222
C04484=1051.841,419.576,372.051,175.090,41.827,158.219
C04485=1051.832,419.330,372.099,175.081,41.818,158.216
C04486=1051.823,419.085,372.145,175.071,41.809,158.213
C04487=1051.813,418.839,372.192,175.062,41.800,158.210
C04488=1051.803,418.593,372.238,175.052,41.792,158.208
C04489=1051.788,418.217,372.309,175.037,41.779,158.203
C04490=1051.773,417.841,372.381,175.023,41.765,158.199
C04491=1051.758,417.464,372.452,175.009,41.752,158.195
C04492=1051.743,417.087,372.523,174.995,41.739,158.190
C04493=1051.734,416.842,372.569,174.985,41.730,158.187
C04494=1051.725,416.597,372.615,174.976,41.722,158.185
C04495=1051.715,416.351,372.662,174.967,41.713,158.182
C04496=1051.706,416.105,372.707,174.958,41.705,158.179
C04497=1051.696,415.859,372.754,174.948,41.696,158.176
C04498=1051.687,415.614,372.800,174.940,41.688,158.173
C04499=1051.677,415.369,372.846,174.931,41.679,158.171
C04500=1051.668,415.123,372.893,174.922,41.671,158.168
C04501=1051.659,414.877,372.938,174.912,41.663,158.165
C04502=1051.649,414.632,372.984,174.904,41.654,158.163
C04503=1051.640,414.386,373.030,174.895,41.645,158.160
C04504=1051.631,414.141,373.076,174.886,41.637,158.157
C04505=1051.621,413.895,373.122,174.877,41.629,158.154
C04506=1051.612,413.649,373.168,174.869,41.621,158.152
C04507=1051.603,413.403,373.213,174.859,41.612,158.149
C04508=1051.594,413.158,373.259,174.850,41.604,158.146
C04509=1051.584,412.912,373.304,174.842,41.596,158.144
C04510=1051.575,412.666,373.350,174.833,41.588,158.141
C04511=1051.565,412.421,373.396,174.824,41.580,158.139
C04512=1051.556,412.175,373.441,174.816,41.571,158.136
C04513=1051.547,411.929,373.486,174.807,41.563,158.133
C04514=1051.538,411.684,373.532,174.798,41.555,158.131
C04515=1051.528,411.438,373.576,174.790,41.547,158.128
C04516=1051.519,411.192,373.622,174.781,41.539,158.126
C04517=1051.509,410.947,373.667,174.773,41.531,158.123
C04518=1051.500,410.701,373.712,174.764,41.524,158.121
C04519=1051.491,410.455,373.758,174.755,41.516,158.118
C04520=1051.482,410.209,373.802,174.747,41.507,158.115
C04521=1051.473,409.964,373.848,174.738,41.500,158.113
C04522=1051.463,409.718,373.893,174.730,41.492,158.110
C04523=1051.454,409.472,373.937,174.721,41.484,158.108
C04524=1051.445,409.226,373.983,174.713,41.476,158.105
C04525=1051.436,408.980,374.028,174.704,41.468,158.103
C04526=1051.427,408.735,374.073,174.697,41.460,158.100
C04527=1051.417,408.488,374.117,174.689,41.452,158.098
C04528=1051.409,408.243,374.162,174.680,41.445,158.095
C04529=1051.400,407.997,374.207,174.672,41.437,158.093
C04530=1051.390,407.751,374.252,174.663,41.429,158.090
C04531=1051.382,407.505,374.296,174.655,41.421,158.088
C04532=1051.373,407.260,374.341,174.647,41.414,158.086
C04533=1051.364,407.014,374.386,174.639,41.406,158.083
C04534=1051.354,406.768,374.430,174.631,41.399,158.081
C04535=1051.346,406.522,374.475,174.623,41.391,158.078
C04536=1051.336,406.277,374.519,174.614,41.383,158.076
C04537=1051.328,406.030,374.564,174.607,41.376,158.074
C04538=1051.320,405.785,374.609,174.599,41.368,158.071
C04539=1051.310,405.539,374.653,174.590,41.360,158.069
C04540=1051.302,405.293,374.698,174.582,41.353,158.066
C04541=1051.292,405.047,374.742,174.575,41.345,158.064
C04542=1051.284,404.801,374.787,174.567,41.338,158.062
C04543=1051.275,404.555,374.830,174.558,41.330,158.059
C04544=1051.266,404.309,374.874,174.550,41.323,158.057
C04545=1051.253,403.939,374.941,174.538,41.312,158.053
C04546=1051.239,403.570,375.007,174.528,41.301,158.050
C04547=1051.226,403.199,375.074,174.516,41.290,158.047
C04548=1051.213,402.829,375.139,174.504,41.278,158.043
C04549=1051.204,402.583,375.184,174.496,41.271,158.041
C04550=1051.196,402.337,375.228,174.488,41.264,158.039
C04551=1051.187,402.092,375.271,174.481,41.256,158.036
C04552=1051.178,401.845,375.315,174.473,41.249,158.034
C04553=1051.170,401.599,375.359,174.465,41.242,158.032
C04554=1051.160,401.353,375.403,174.457,41.235,158.029
C04555=1051.152,401.107,375.446,174.449,41.228,158.027
C04556=1051.143,400.862,375.490,174.442,41.221,158.025
C04557=1051.134,400.615,375.533,174.434,41.213,158.023
C04558=1051.125,400.370,375.577,174.427,41.206,158.021
C04559=1051.116,400.124,375.620,174.419,41.199,158.018
C04560=1051.108,399.878,375.665,174.412,41.193,158.016
C04561=1051.099,399.631,375.708,174.404,41.185,158.014
C04562=1051.091,399.385,375.751,174.397,41.178,158.012
C04563=1051.082,399.140,375.795,174.389,41.171,158.010
C04564=1051.073,398.894,375.838,174.382,41.164,158.008
C04565=1051.065,398.648,375.881,174.375,41.157,158.005
C04566=1051.056,398.401,375.924,174.367,41.150,158.003
C04567=1051.047,398.155,375.968,174.360,41.143,158.001
C04568=1051.039,397.909,376.011,174.352,41.136,157.999
C04569=1051.030,397.663,376.054,174.345,41.129,157.997
C04570=1051.022,397.417,376.097,174.337,41.122,157.995
C04571=1051.013,397.171,376.140,174.330,41.116,157.993
C04572=1051.005,396.925,376.183,174.323,41.109,157.990
C04573=1050.996,396.679,376.226,174.315,41.102,157.988
C04574=1050.988,396.433,376.269,174.309,41.095,157.986
C04575=1050.979,396.187,376.312,174.302,41.088,157.984
C04576=1050.971,395.941,376.355,174.294,41.082,157.982
C04577=1050.962,395.695,376.398,174.287,41.074,157.980
C04578=1050.954,395.449,376.441,174.280,41.068,157.978
C04579=1050.945,395.202,376.483,174.272,41.061,157.976
C04580=1050.936,394.956,376.526,174.265,41.054,157.974
C04581=1050.928,394.710,376.569,174.258,41.048,157.972
C04582=1050.919,394.464,376.612,174.251,41.041,157.970
C04583=1050.911,394.218,376.654,174.244,41.034,157.968
C04584=1050.903,393.972,376.697,174.237,41.028,157.966
C04585=1050.895,393.725,376.739,174.230,41.021,157.964
C04586=1050.886,393.479,376.782,174.222,41.015,157.962
C04587=1050.877,393.234,376.825,174.216,41.008,157.960
C04588=1050.869,392.988,376.867,174.209,41.001,157.958
C04589=1050.859,392.679,376.921,174.200,40.993,157.955
C04590=1050.848,392.369,376.973,174.191,40.985,157.952
C04591=1050.838,392.060,377.027,174.182,40.976,157.950
C04592=1050.827,391.752,377.080,174.174,40.969,157.948
C04593=1050.819,391.505,377.122,174.166,40.962,157.946
C04594=1050.810,391.259,377.164,174.160,40.956,157.944
C04595=1050.802,391.013,377.207,174.153,40.949,157.942
C04596=1050.793,390.767,377.248,174.146,40.943,157.940
C04597=1050.785,390.520,377.291,174.139,40.936,157.938
C04598=1050.778,390.274,377.333,174.133,40.930,157.936
C04599=1050.769,390.028,377.374,174.125,40.924,157.934
C04600=1050.760,389.782,377.417,174.119,40.917,157.932
C04601=1050.751,389.493,377.466,174.111,40.910,157.930
C04602=1050.741,389.204,377.515,174.103,40.902,157.928
C04603=1050.732,388.915,377.564,174.095,40.895,157.925
C04604=1050.721,388.626,377.614,174.087,40.887,157.923
C04605=1050.713,388.380,377.655,174.080,40.881,157.921
C04606=1050.705,388.134,377.697,174.073,40.875,157.919
C04607=1050.697,387.888,377.739,174.067,40.869,157.917
C04608=1050.689,387.641,377.780,174.060,40.863,157.916
C04609=1050.680,387.395,377.822,174.054,40.857,157.914
C04610=1050.671,387.149,377.863,174.047,40.851,157.912
C04611=1050.664,386.903,377.905,174.041,40.844,157.910
C04612=1050.655,386.656,377.946,174.034,40.838,157.908
C04613=1050.648,386.410,377.988,174.027,40.832,157.906
C04614=1050.639,386.163,378.030,174.021,40.826,157.905
C04615=1050.631,385.917,378.070,174.014,40.820,157.903
C04616=1050.622,385.671,378.113,174.008,40.814,157.901
C04617=1050.614,385.424,378.153,174.001,40.808,157.899
C04618=1050.605,385.178,378.195,173.995,40.802,157.897
C04619=1050.598,384.931,378.236,173.988,40.796,157.895
C04620=1050.590,384.686,378.278,173.982,40.790,157.894
C04621=1050.581,384.439,378.319,173.975,40.784,157.892
C04622=1050.574,384.193,378.361,173.969,40.778,157.890
C04623=1050.566,383.946,378.401,173.962,40.772,157.888
C04624=1050.557,383.699,378.442,173.956,40.766,157.887
C04625=1050.549,383.453,378.484,173.950,40.760,157.885
C04626=1050.541,383.207,378.525,173.943,40.754,157.883
C04627=1050.533,382.960,378.566,173.937,40.748,157.881
C04628=1050.525,382.714,378.607,173.930,40.742,157.879
C04629=1050.517,382.468,378.648,173.924,40.736,157.878
C04630=1050.509,382.222,378.689,173.917,40.730,157.876
C04631=1050.502,381.975,378.730,173.911,40.724,157.874
C04632=1050.493,381.728,378.771,173.906,40.718,157.872
C04633=1050.485,381.482,378.812,173.899,40.713,157.871
C04634=1050.478,381.235,378.853,173.893,40.707,157.869
C04635=1050.470,380.989,378.894,173.887,40.701,157.867
C04636=1050.462,380.743,378.934,173.880,40.695,157.865
C04637=1050.454,380.496,378.976,173.874,40.689,157.864
C04638=1050.446,380.249,379.017,173.868,40.683,157.862
C04639=1050.438,380.003,379.057,173.861,40.678,157.860
C04640=1050.430,379.756,379.098,173.856,40.672,157.859
C04641=1050.423,379.510,379.139,173.850,40.666,157.857
C04642=1050.414,379.264,379.180,173.843,40.660,157.855
C04643=1050.406,379.017,379.220,173.837,40.655,157.854
C04644=1050.398,378.771,379.260,173.831,40.649,157.852
C04645=1050.390,378.524,379.300,173.824,40.644,157.850
C04646=1050.382,378.278,379.341,173.819,40.638,157.849
C04647=1050.374,378.031,379.381,173.813,40.632,157.847
C04648=1050.366,377.785,379.422,173.806,40.627,157.845
C04649=1050.358,377.538,379.463,173.800,40.621,157.844
C04650=1050.350,377.291,379.503,173.794,40.615,157.842
C04651=1050.342,377.045,379.543,173.789,40.610,157.840
C04652=1050.334,376.798,379.583,173.782,40.604,157.839
C04653=1050.326,376.552,379.624,173.776,40.599,157.837
C04654=1050.318,376.305,379.664,173.770,40.593,157.836
C04655=1050.310,376.058,379.704,173.765,40.588,157.834
C04656=1050.303,375.812,379.744,173.759,40.582,157.832
C04657=1050.293,375.493,379.796,173.751,40.575,157.830
C04658=1050.283,375.173,379.848,173.743,40.568,157.828
C04659=1050.273,374.854,379.900,173.735,40.561,157.826
C04660=1050.263,374.536,379.952,173.728,40.554,157.824
C04661=1050.255,374.289,379.992,173.722,40.548,157.822
C04662=1050.247,374.042,380.032,173.717,40.543,157.821
C04663=1050.240,373.795,380.072,173.710,40.538,157.819
C04664=1050.232,373.548,380.112,173.704,40.532,157.818
C04665=1050.223,373.302,380.151,173.698,40.527,157.816
C04666=1050.216,373.056,380.191,173.693,40.521,157.814
C04667=1050.208,372.809,380.231,173.687,40.516,157.813
C04668=1050.200,372.563,380.272,173.681,40.510,157.811
C04669=1050.193,372.316,380.311,173.676,40.505,157.810
C04670=1050.186,372.069,380.351,173.670,40.500,157.808
C04671=1050.178,371.823,380.391,173.663,40.495,157.807
C04672=1050.170,371.576,380.431,173.658,40.489,157.805
C04673=1050.162,371.329,380.471,173.652,40.484,157.804
C04674=1050.155,371.082,380.509,173.646,40.479,157.802
C04675=1050.147,370.835,380.549,173.641,40.474,157.801
C04676=1050.139,370.588,380.589,173.635,40.468,157.799
C04677=1050.131,370.342,380.628,173.630,40.463,157.797
C04678=1050.124,370.096,380.668,173.624,40.458,157.796
C04679=1050.116,369.848,380.706,173.618,40.452,157.794
C04680=1050.108,369.601,380.746,173.613,40.448,157.793
C04681=1050.101,369.355,380.786,173.607,40.442,157.792
C04682=1050.093,369.108,380.824,173.602,40.437,157.790
C04683=1050.085,368.861,380.864,173.596,40.432,157.788
C04684=1050.077,368.615,380.903,173.590,40.427,157.787
C04685=1050.070,368.368,380.942,173.585,40.422,157.786
C04686=1050.062,368.121,380.982,173.579,40.416,157.784
C04687=1050.054,367.875,381.021,173.574,40.412,157.783
C04688=1050.047,367.627,381.061,173.568,40.406,157.781
C04689=1050.039,367.381,381.100,173.563,40.401,157.780
C04690=1050.032,367.134,381.139,173.557,40.396,157.778
C04691=1050.024,366.888,381.178,173.551,40.391,157.777
C04692=1050.016,366.641,381.217,173.546,40.386,157.775
C04693=1050.008,366.393,381.255,173.540,40.381,157.774
C04694=1050.001,366.147,381.295,173.535,40.376,157.772
C04695=1049.994,365.900,381.334,173.529,40.371,157.771
C04696=1049.986,365.653,381.372,173.524,40.366,157.769
C04697=1049.979,365.407,381.412,173.518,40.361,157.768
C04698=1049.971,365.160,381.451,173.513,40.356,157.767
C04699=1049.964,364.913,381.489,173.507,40.351,157.765
C04700=1049.955,364.666,381.529,173.502,40.346,157.764
C04701=1049.949,364.419,381.568,173.496,40.341,157.762
C04702=1049.941,364.172,381.606,173.491,40.336,157.761
C04703=1049.934,363.925,381.645,173.486,40.331,157.760
C04704=1049.926,363.679,381.683,173.481,40.326,157.758
C04705=1049.918,363.432,381.723,173.475,40.321,157.757
C04706=1049.912,363.185,381.762,173.470,40.316,157.755
C04707=1049.903,362.938,381.801,173.464,40.311,157.754
C04708=1049.896,362.691,381.839,173.459,40.306,157.752
C04709=1049.889,362.445,381.878,173.453,40.302,157.751
C04710=1049.881,362.197,381.916,173.448,40.297,157.750
C04711=1049.873,361.951,381.955,173.443,40.292,157.748
C04712=1049.866,361.704,381.993,173.438,40.287,157.747
C04713=1049.856,361.404,382.040,173.431,40.281,157.745
C04714=1049.848,361.103,382.086,173.424,40.276,157.744
C04715=1049.839,360.803,382.133,173.419,40.270,157.742
C04716=1049.829,360.503,382.179,173.412,40.264,157.740
C04717=1049.822,360.257,382.218,173.407,40.259,157.739
C04718=1049.815,360.010,382.256,173.401,40.254,157.738
C04719=1049.807,359.762,382.294,173.397,40.250,157.736
C04720=1049.800,359.516,382.332,173.391,40.245,157.735
C04721=1049.793,359.269,382.371,173.386,40.240,157.734
C04722=1049.785,359.022,382.410,173.380,40.235,157.732
C04723=1049.777,358.775,382.447,173.376,40.231,157.731
C04724=1049.770,358.528,382.486,173.371,40.226,157.730
C04725=1049.763,358.281,382.523,173.365,40.221,157.728
C04726=1049.756,358.034,382.562,173.360,40.217,157.727
C04727=1049.748,357.788,382.600,173.356,40.212,157.726
C04728=1049.740,357.540,382.638,173.350,40.208,157.724
C04729=1049.733,357.293,382.676,173.345,40.203,157.723
C04730=1049.726,357.046,382.714,173.339,40.198,157.722
C04731=1049.718,356.799,382.751,173.335,40.194,157.720
C04732=1049.711,356.552,382.790,173.330,40.189,157.719
C04733=1049.703,356.305,382.827,173.324,40.184,157.718
C04734=1049.695,356.058,382.866,173.319,40.180,157.716
C04735=1049.688,355.811,382.903,173.315,40.175,157.715
C04736=1049.681,355.564,382.941,173.309,40.171,157.714
C04737=1049.674,355.317,382.978,173.304,40.166,157.713
C04738=1049.666,355.070,383.017,173.300,40.162,157.711
C04739=1049.659,354.823,383.054,173.294,40.157,157.710
C04740=1049.652,354.576,383.092,173.289,40.153,157.709
C04741=1049.644,354.329,383.129,173.284,40.148,157.707
C04742=1049.637,354.082,383.167,173.279,40.144,157.706
C04743=1049.630,353.835,383.205,173.274,40.139,157.705
C04744=1049.622,353.588,383.243,173.270,40.134,157.704
C04745=1049.615,353.341,383.280,173.264,40.130,157.702
C04746=1049.608,353.094,383.318,173.259,40.125,157.701
C04747=1049.601,352.847,383.355,173.255,40.121,157.700
C04748=1049.593,352.599,383.393,173.250,40.116,157.699
C04749=1049.586,352.352,383.430,173.244,40.112,157.697
C04750=1049.579,352.105,383.468,173.240,40.108,157.696
C04751=1049.572,351.858,383.505,173.235,40.103,157.695
C04752=1049.564,351.611,383.543,173.229,40.099,157.694
C04753=1049.557,351.364,383.580,173.225,40.094,157.692
C04754=1049.550,351.117,383.618,173.220,40.090,157.691
C04755=1049.543,350.869,383.655,173.216,40.085,157.690
C04756=1049.535,350.623,383.692,173.210,40.081,157.689
C04757=1049.527,350.376,383.730,173.206,40.077,157.688
C04758=1049.521,350.129,383.767,173.201,40.072,157.686
C04759=1049.514,349.881,383.804,173.196,40.068,157.685
C04760=1049.506,349.635,383.841,173.191,40.064,157.684
C04761=1049.499,349.387,383.878,173.186,40.059,157.683
C04762=1049.492,349.140,383.915,173.182,40.055,157.681
C04763=1049.484,348.892,383.953,173.177,40.050,157.680
C04764=1049.476,348.646,383.989,173.171,40.046,157.679
C04765=1049.469,348.399,384.027,173.167,40.042,157.678
C04766=1049.463,348.151,384.063,173.162,40.038,157.677
C04767=1049.455,347.905,384.100,173.158,40.033,157.675
C04768=1049.448,347.657,384.137,173.152,40.029,157.674
C04769=1049.439,347.363,384.182,173.147,40.024,157.673
C04770=1049.431,347.068,384.226,173.141,40.019,157.671
C04771=1049.422,346.773,384.270,173.136,40.014,157.670
C04772=1049.414,346.478,384.314,173.131,40.008,157.669
C04773=1049.406,346.231,384.351,173.125,40.005,157.667
C04774=1049.399,345.984,384.387,173.121,40.000,157.666
C04775=1049.392,345.737,384.425,173.116,39.996,157.665
C04776=1049.385,345.490,384.461,173.112,39.992,157.664
C04777=1049.378,345.242,384.498,173.107,39.988,157.663
C04778=1049.371,344.995,384.535,173.102,39.983,157.662
C04779=1049.363,344.748,384.571,173.097,39.980,157.660
C04780=1049.357,344.500,384.608,173.093,39.975,157.659
C04781=1049.349,344.253,384.645,173.088,39.971,157.658
C04782=1049.342,344.006,384.681,173.084,39.967,157.657
C04783=1049.335,343.759,384.718,173.079,39.963,157.656
C04784=1049.328,343.511,384.754,173.074,39.959,157.655
C04785=1049.321,343.265,384.791,173.069,39.954,157.653
C04786=1049.313,343.017,384.828,173.065,39.950,157.652
C04787=1049.307,342.770,384.864,173.061,39.946,157.651
C04788=1049.299,342.523,384.900,173.056,39.942,157.650
C04789=1049.292,342.275,384.937,173.052,39.938,157.649
C04790=1049.285,342.028,384.973,173.046,39.934,157.648
C04791=1049.278,341.781,385.010,173.042,39.930,157.647
C04792=1049.271,341.534,385.045,173.038,39.926,157.646
C04793=1049.264,341.286,385.082,173.033,39.922,157.645
C04794=1049.257,341.039,385.119,173.029,39.918,157.643
C04795=1049.250,340.792,385.154,173.024,39.914,157.642
C04796=1049.242,340.544,385.191,173.020,39.909,157.641
C04797=1049.236,340.297,385.227,173.016,39.906,157.640
C04798=1049.228,340.050,385.263,173.010,39.901,157.639
C04799=1049.221,339.803,385.299,173.006,39.898,157.638
C04800=1049.214,339.555,385.336,173.001,39.893,157.637
C04801=1049.207,339.309,385.372,172.997,39.890,157.636
C04802=1049.199,339.061,385.408,172.993,39.886,157.635
C04803=1049.193,338.814,385.444,172.988,39.881,157.633
C04804=1049.185,338.566,385.480,172.984,39.878,157.632
C04805=1049.178,338.319,385.516,172.980,39.873,157.631
C04806=1049.171,338.072,385.553,172.975,39.870,157.630
C04807=1049.164,337.825,385.588,172.971,39.866,157.629
C04808=1049.157,337.577,385.624,172.966,39.861,157.628
C04809=1049.151,337.330,385.660,172.961,39.858,157.627
C04810=1049.143,337.082,385.697,172.957,39.854,157.626
C04811=1049.136,336.835,385.732,172.953,39.849,157.625
C04812=1049.129,336.588,385.768,172.948,39.846,157.624
C04813=1049.122,336.340,385.804,172.944,39.842,157.623
C04814=1049.115,336.093,385.840,172.940,39.838,157.622
C04815=1049.108,335.846,385.876,172.936,39.834,157.620
C04816=1049.101,335.598,385.911,172.931,39.830,157.619
C04817=1049.094,335.352,385.947,172.927,39.826,157.618
C04818=1049.086,335.103,385.982,172.923,39.822,157.617
C04819=1049.080,334.856,386.019,172.918,39.819,157.616
C04820=1049.073,334.608,386.054,172.914,39.815,157.615
C04821=1049.066,334.362,386.090,172.909,39.811,157.614
C04822=1049.059,334.114,386.125,172.904,39.807,157.613
C04823=1049.052,333.866,386.161,172.900,39.804,157.612
C04824=1049.044,333.619,386.197,172.896,39.799,157.611
C04825=1049.036,333.321,386.239,172.891,39.795,157.610
C04826=1049.028,333.023,386.282,172.886,39.790,157.608
C04827=1049.019,332.724,386.325,172.881,39.786,157.607
C04828=1049.011,332.425,386.367,172.875,39.781,157.606
C04829=1049.004,332.178,386.403,172.871,39.778,157.605
C04830=1048.996,331.930,386.439,172.867,39.774,157.604
C04831=1048.990,331.683,386.474,172.863,39.770,157.603
C04832=1048.983,331.435,386.509,172.858,39.766,157.602
C04833=1048.976,331.189,386.545,172.854,39.762,157.601
C04834=1048.969,330.941,386.580,172.850,39.759,157.600
C04835=1048.962,330.693,386.615,172.846,39.755,157.599
C04836=1048.955,330.446,386.651,172.842,39.751,157.598
C04837=1048.948,330.198,386.686,172.837,39.747,157.597
C04838=1048.941,329.951,386.721,172.833,39.743,157.596
C04839=1048.935,329.704,386.756,172.829,39.739,157.595
C04840=1048.927,329.456,386.792,172.825,39.736,157.594
C04841=1048.921,329.208,386.827,172.821,39.732,157.593
C04842=1048.913,328.961,386.861,172.817,39.729,157.592
C04843=1048.906,328.714,386.896,172.812,39.725,157.591
C04844=1048.899,328.466,386.932,172.808,39.721,157.590
C04845=1048.891,328.219,386.966,172.804,39.718,157.589
C04846=1048.885,327.971,387.002,172.800,39.714,157.588
C04847=1048.878,327.724,387.037,172.796,39.710,157.587
C04848=1048.870,327.477,387.071,172.791,39.707,157.586
C04849=1048.864,327.230,387.106,172.787,39.703,157.585
C04850=1048.856,326.981,387.141,172.783,39.700,157.584
C04851=1048.849,326.734,387.176,172.779,39.696,157.583
C04852=1048.842,326.486,387.211,172.775,39.692,157.582
C04853=1048.835,326.239,387.245,172.771,39.689,157.581
C04854=1048.828,325.991,387.280,172.766,39.685,157.580
C04855=1048.821,325.744,387.315,172.763,39.682,157.579
C04856=1048.814,325.497,387.349,172.759,39.678,157.578
C04857=1048.807,325.250,387.385,172.755,39.674,157.577
C04858=1048.801,325.002,387.419,172.751,39.671,157.576
C04859=1048.793,324.754,387.454,172.747,39.667,157.575
C04860=1048.786,324.507,387.489,172.743,39.664,157.574
C04861=1048.779,324.259,387.523,172.739,39.660,157.573
C04862=1048.772,324.012,387.558,172.735,39.657,157.572
C04863=1048.765,323.764,387.592,172.730,39.653,157.571
C04864=1048.758,323.516,387.627,172.726,39.650,157.571
C04865=1048.751,323.268,387.661,172.722,39.646,157.570
C04866=1048.744,323.021,387.696,172.718,39.643,157.569
C04867=1048.737,322.774,387.731,172.714,39.639,157.568
C04868=1048.730,322.526,387.765,172.710,39.636,157.567
C04869=1048.723,322.279,387.800,172.706,39.632,157.566
C04870=1048.717,322.032,387.834,172.702,39.628,157.565
C04871=1048.710,321.784,387.868,172.698,39.625,157.564
C04872=1048.703,321.537,387.903,172.695,39.621,157.563
C04873=1048.696,321.289,387.937,172.691,39.617,157.562
C04874=1048.689,321.042,387.972,172.687,39.614,157.561
C04875=1048.682,320.794,388.006,172.683,39.611,157.560
C04876=1048.675,320.547,388.041,172.679,39.607,157.559
C04877=1048.669,320.299,388.075,172.675,39.604,157.558
C04878=1048.662,320.051,388.109,172.671,39.600,157.557
C04879=1048.656,319.804,388.144,172.667,39.597,157.556
C04880=1048.648,319.557,388.178,172.663,39.593,157.556
C04881=1048.640,319.253,388.220,172.658,39.589,157.554
C04882=1048.632,318.949,388.262,172.653,39.585,157.553
C04883=1048.623,318.645,388.304,172.649,39.580,157.552
C04884=1048.615,318.342,388.346,172.644,39.576,157.551
C04885=1048.609,318.094,388.380,172.640,39.573,157.550
C04886=1048.601,317.847,388.415,172.636,39.569,157.549
C04887=1048.595,317.599,388.449,172.632,39.565,157.548
C04888=1048.588,317.351,388.483,172.628,39.562,157.547
C04889=1048.582,317.104,388.517,172.624,39.559,157.546
C04890=1048.575,316.856,388.551,172.620,39.555,157.545
C04891=1048.568,316.608,388.585,172.616,39.552,157.545
C04892=1048.561,316.362,388.619,172.613,39.548,157.544
C04893=1048.555,316.114,388.654,172.609,39.545,157.543
C04894=1048.548,315.866,388.688,172.605,39.541,157.542
C04895=1048.541,315.618,388.722,172.602,39.538,157.541
C04896=1048.535,315.371,388.755,172.598,39.535,157.540
C04897=1048.528,315.123,388.790,172.594,39.531,157.539
C04898=1048.521,314.876,388.824,172.590,39.527,157.538
C04899=1048.515,314.628,388.858,172.586,39.524,157.537
C04900=1048.508,314.381,388.892,172.582,39.521,157.536
C04901=1048.502,314.133,388.926,172.579,39.518,157.536
C04902=1048.495,313.886,388.959,172.575,39.514,157.535
C04903=1048.488,313.638,388.994,172.571,39.510,157.534
C04904=1048.482,313.391,389.027,172.567,39.507,157.533
C04905=1048.475,313.143,389.062,172.564,39.504,157.532
C04906=1048.469,312.895,389.094,172.560,39.500,157.531
C04907=1048.462,312.647,389.128,172.556,39.497,157.530
C04908=1048.455,312.400,389.162,172.553,39.494,157.529
C04909=1048.448,312.153,389.196,172.549,39.491,157.528
C04910=1048.441,311.905,389.229,172.545,39.487,157.528
C04911=1048.434,311.657,389.263,172.541,39.484,157.527
C04912=1048.427,311.410,389.296,172.537,39.481,157.526
C04913=1048.420,311.162,389.329,172.533,39.477,157.525
C04914=1048.413,310.914,389.363,172.530,39.474,157.524
C04915=1048.407,310.666,389.396,172.526,39.471,157.523
C04916=1048.399,310.419,389.429,172.523,39.467,157.522
C04917=1048.392,310.171,389.463,172.519,39.464,157.521
C04918=1048.385,309.924,389.495,172.515,39.461,157.521
C04919=1048.378,309.676,389.529,172.511,39.458,157.520
C04920=1048.372,309.428,389.562,172.508,39.455,157.519
C04921=1048.365,309.181,389.596,172.504,39.452,157.518
C04922=1048.358,308.932,389.629,172.500,39.448,157.517
C04923=1048.351,308.685,389.662,172.496,39.445,157.516
C04924=1048.344,308.437,389.696,172.493,39.442,157.516
C04925=1048.338,308.190,389.729,172.489,39.438,157.515
C04926=1048.331,307.942,389.762,172.486,39.436,157.514
C04927=1048.324,307.695,389.795,172.482,39.432,157.513
C04928=1048.317,307.447,389.828,172.478,39.429,157.512
C04929=1048.310,307.200,389.862,172.474,39.426,157.511
C04930=1048.303,306.952,389.895,172.470,39.422,157.511
C04931=1048.297,306.704,389.927,172.468,39.419,157.510
C04932=1048.290,306.456,389.961,172.464,39.416,157.509
C04933=1048.283,306.209,389.994,172.460,39.413,157.508
C04934=1048.276,305.961,390.027,172.456,39.410,157.507
C04935=1048.269,305.714,390.060,172.452,39.406,157.506
C04936=1048.263,305.466,390.093,172.450,39.404,157.506
C04937=1048.254,305.167,390.132,172.445,39.400,157.505
C04938=1048.247,304.868,390.173,172.441,39.396,157.504
C04939=1048.238,304.568,390.213,172.436,39.392,157.503
C04940=1048.230,304.269,390.252,172.432,39.388,157.502
C04941=1048.224,304.021,390.285,172.428,39.385,157.501
C04942=1048.217,303.773,390.318,172.425,39.381,157.500
C04943=1048.211,303.526,390.352,172.421,39.378,157.499
C04944=1048.203,303.278,390.384,172.418,39.375,157.498
C04945=1048.197,303.031,390.417,172.414,39.372,157.497
C04946=1048.190,302.783,390.450,172.411,39.369,157.497
C04947=1048.184,302.535,390.483,172.407,39.365,157.496
C04948=1048.177,302.287,390.515,172.403,39.363,157.495
C04949=1048.171,302.040,390.548,172.400,39.359,157.494
C04950=1048.163,301.792,390.581,172.397,39.356,157.493
C04951=1048.157,301.545,390.614,172.393,39.353,157.493
C04952=1048.150,301.297,390.647,172.389,39.350,157.492
C04953=1048.144,301.049,390.680,172.385,39.347,157.491
C04954=1048.137,300.801,390.713,172.383,39.343,157.490
C04955=1048.130,300.554,390.745,172.379,39.340,157.489
C04956=1048.124,300.306,390.778,172.375,39.337,157.488
C04957=1048.117,300.058,390.811,172.372,39.334,157.488
C04958=1048.111,299.810,390.844,172.369,39.331,157.487
C04959=1048.104,299.563,390.876,172.365,39.328,157.486
C04960=1048.098,299.315,390.908,172.362,39.324,157.485
C04961=1048.091,299.067,390.940,172.358,39.322,157.484
C04962=1048.085,298.819,390.974,172.354,39.318,157.484
C04963=1048.078,298.571,391.006,172.352,39.315,157.483
C04964=1048.072,298.324,391.039,172.348,39.312,157.482
C04965=1048.066,298.076,391.072,172.344,39.309,157.481
C04966=1048.059,297.829,391.104,172.341,39.305,157.480
C04967=1048.052,297.581,391.137,172.338,39.303,157.480
C04968=1048.046,297.332,391.169,172.334,39.299,157.479
C04969=1048.039,297.085,391.202,172.331,39.296,157.478
C04970=1048.032,296.838,391.234,172.327,39.293,157.477
C04971=1048.026,296.590,391.267,172.324,39.290,157.476
C04972=1048.020,296.342,391.299,172.321,39.287,157.476
C04973=1048.014,296.094,391.331,172.317,39.284,157.475
C04974=1048.006,295.846,391.364,172.313,39.280,157.474
C04975=1048.000,295.598,391.396,172.311,39.277,157.473
C04976=1047.993,295.351,391.428,172.307,39.274,157.472
C04977=1047.987,295.103,391.461,172.303,39.271,157.472
C04978=1047.980,294.855,391.492,172.300,39.268,157.471
C04979=1047.974,294.608,391.525,172.297,39.265,157.470
C04980=1047.967,294.359,391.557,172.294,39.262,157.469
C04981=1047.960,294.111,391.590,172.290,39.259,157.468
C04982=1047.953,293.864,391.622,172.286,39.256,157.468
C04983=1047.947,293.616,391.653,172.284,39.253,157.467
C04984=1047.941,293.368,391.685,172.280,39.250,157.466
C04985=1047.934,293.121,391.717,172.276,39.247,157.465
C04986=1047.928,292.873,391.749,172.273,39.244,157.465
C04987=1047.920,292.625,391.782,172.270,39.241,157.464
C04988=1047.913,292.377,391.813,172.267,39.238,157.463
C04989=1047.907,292.129,391.846,172.263,39.235,157.462
C04990=1047.900,291.881,391.878,172.260,39.232,157.462
C04991=1047.893,291.633,391.909,172.257,39.229,157.461
C04992=1047.887,291.386,391.942,172.253,39.226,157.460
C04993=1047.879,291.103,391.978,172.249,39.223,157.459
C04994=1047.872,290.819,392.014,172.246,39.220,157.458
C04995=1047.864,290.536,392.051,172.242,39.216,157.457
C04996=1047.857,290.254,392.087,172.239,39.212,157.456
C04997=1047.851,290.006,392.119,172.235,39.209,157.456
C04998=1047.844,289.758,392.150,172.231,39.207,157.455
C04999=1047.837,289.511,392.182,172.229,39.203,157.454
C05000=1047.831,289.262,392.214,172.225,39.201,157.453
C05001=1047.824,289.014,392.246,172.222,39.198,157.453
C05002=1047.817,288.767,392.277,172.219,39.194,157.452
C05003=1047.810,288.519,392.309,172.216,39.192,157.451
C05004=1047.804,288.271,392.341,172.212,39.189,157.450
C05005=1047.798,288.023,392.373,172.209,39.185,157.450
C05006=1047.791,287.775,392.404,172.206,39.183,157.449
C05007=1047.784,287.527,392.436,172.202,39.180,157.448
C05008=1047.777,287.279,392.467,172.199,39.177,157.448
C05009=1047.771,287.032,392.499,172.196,39.174,157.447
C05010=1047.764,286.784,392.530,172.193,39.171,157.446
C05011=1047.758,286.535,392.562,172.189,39.168,157.445
C05012=1047.751,286.288,392.593,172.187,39.165,157.445
C05013=1047.745,286.040,392.625,172.183,39.162,157.444
C05014=1047.738,285.792,392.656,172.180,39.159,157.443
C05015=1047.731,285.544,392.688,172.176,39.156,157.442
C05016=1047.724,285.296,392.719,172.174,39.153,157.442
C05017=1047.718,285.048,392.751,172.170,39.151,157.441
C05018=1047.711,284.800,392.782,172.167,39.148,157.440
C05019=1047.704,284.552,392.813,172.164,39.144,157.439
C05020=1047.698,284.304,392.845,172.161,39.142,157.439
C05021=1047.691,284.056,392.876,172.157,39.139,157.438
C05022=1047.684,283.808,392.908,172.155,39.136,157.437
C05023=1047.677,283.561,392.939,172.151,39.133,157.436
C05024=1047.672,283.313,392.970,172.148,39.130,157.436
C05025=1047.665,283.065,393.001,172.145,39.127,157.435
C05026=1047.658,282.817,393.032,172.142,39.124,157.434
C05027=1047.651,282.569,393.064,172.138,39.121,157.434
C05028=1047.645,282.321,393.095,172.136,39.119,157.433
C05029=1047.638,282.073,393.127,172.133,39.116,157.432
C05030=1047.631,281.825,393.157,172.129,39.112,157.431
C05031=1047.625,281.578,393.188,172.127,39.110,157.431
C05032=1047.619,281.330,393.220,172.123,39.107,157.430
C05033=1047.612,281.082,393.251,172.120,39.104,157.429
C05034=1047.605,280.833,393.282,172.117,39.101,157.428
C05035=1047.599,280.585,393.314,172.114,39.098,157.428
C05036=1047.593,280.338,393.345,172.110,39.095,157.427
C05037=1047.586,280.090,393.375,172.107,39.092,157.426
C05038=1047.579,279.842,393.407,172.105,39.089,157.425
C05039=1047.573,279.594,393.438,172.101,39.087,157.425
C05040=1047.566,279.345,393.469,172.098,39.084,157.424
C05041=1047.560,279.098,393.500,172.095,39.081,157.423
C05042=1047.554,278.850,393.531,172.092,39.078,157.423
C05043=1047.547,278.602,393.562,172.090,39.075,157.422
C05044=1047.541,278.353,393.593,172.086,39.072,157.421
C05045=1047.533,278.105,393.624,172.083,39.070,157.421
C05046=1047.527,277.858,393.655,172.080,39.067,157.420
C05047=1047.521,277.610,393.685,172.077,39.063,157.419
C05048=1047.514,277.361,393.716,172.074,39.061,157.418
C05049=1047.506,277.090,393.750,172.070,39.058,157.418
C05050=1047.500,276.818,393.784,172.067,39.054,157.417
C05051=1047.492,276.547,393.817,172.064,39.052,157.416
C05052=1047.485,276.275,393.851,172.060,39.048,157.415
C05053=1047.478,276.028,393.882,172.058,39.045,157.415
C05054=1047.472,275.780,393.912,172.054,39.043,157.414
C05055=1047.465,275.532,393.944,172.051,39.040,157.413
C05056=1047.460,275.284,393.974,172.049,39.037,157.412
C05057=1047.452,275.036,394.004,172.045,39.034,157.412
C05058=1047.446,274.788,394.036,172.042,39.031,157.411
C05059=1047.439,274.539,394.067,172.040,39.028,157.410
C05060=1047.433,274.292,394.096,172.036,39.026,157.410
C05061=1047.426,274.044,394.128,172.033,39.023,157.409
C05062=1047.420,273.795,394.158,172.030,39.020,157.408
C05063=1047.413,273.548,394.188,172.027,39.017,157.408
C05064=1047.407,273.299,394.219,172.024,39.014,157.407
C05065=1047.400,273.051,394.250,172.021,39.011,157.406
C05066=1047.393,272.804,394.280,172.018,39.009,157.405
C05067=1047.387,272.555,394.311,172.016,39.006,157.405
C05068=1047.381,272.308,394.341,172.013,39.003,157.404
C05069=1047.374,272.059,394.371,172.009,39.000,157.403
C05070=1047.367,271.811,394.403,172.007,38.997,157.403
C05071=1047.361,271.564,394.432,172.004,38.994,157.402
C05072=1047.354,271.315,394.463,172.000,38.992,157.401
C05073=1047.348,271.067,394.494,171.998,38.989,157.401
C05074=1047.341,270.819,394.524,171.995,38.986,157.400
C05075=1047.335,270.571,394.554,171.992,38.984,157.399
C05076=1047.328,270.323,394.585,171.989,38.981,157.399
C05077=1047.322,270.075,394.615,171.986,38.978,157.398
C05078=1047.315,269.827,394.645,171.983,38.975,157.397
C05079=1047.309,269.579,394.675,171.980,38.972,157.396
C05080=1047.302,269.331,394.705,171.977,38.969,157.396
C05081=1047.295,269.082,394.736,171.975,38.967,157.395
C05082=1047.289,268.834,394.766,171.971,38.964,157.394
C05083=1047.282,268.586,394.797,171.968,38.961,157.394
C05084=1047.276,268.338,394.826,171.966,38.958,157.393
C05085=1047.269,268.090,394.857,171.962,38.955,157.392
C05086=1047.263,267.842,394.887,171.960,38.953,157.392
C05087=1047.256,267.594,394.917,171.957,38.950,157.391
C05088=1047.250,267.346,394.947,171.954,38.947,157.390
C05089=1047.243,267.098,394.977,171.951,38.944,157.390
C05090=1047.236,266.850,395.008,171.948,38.942,157.389
C05091=1047.230,266.602,395.037,171.945,38.939,157.388
C05092=1047.223,266.353,395.067,171.943,38.936,157.388
C05093=1047.217,266.105,395.098,171.939,38.933,157.387
C05094=1047.210,265.857,395.128,171.937,38.931,157.386
C05095=1047.203,265.610,395.158,171.934,38.928,157.386
C05096=1047.197,265.361,395.188,171.931,38.925,157.385
C05097=1047.191,265.113,395.217,171.928,38.922,157.384
C05098=1047.183,264.865,395.247,171.925,38.919,157.384
C05099=1047.178,264.617,395.278,171.922,38.917,157.383
C05100=1047.170,264.369,395.308,171.920,38.914,157.382
C05101=1047.164,264.121,395.337,171.916,38.911,157.382
C05102=1047.158,263.872,395.368,171.914,38.909,157.381
C05103=1047.151,263.625,395.397,171.911,38.906,157.380
C05104=1047.144,263.376,395.427,171.908,38.903,157.380
C05105=1047.138,263.109,395.460,171.905,38.900,157.379
C05106=1047.131,262.842,395.491,171.902,38.897,157.378
C05107=1047.124,262.575,395.524,171.899,38.894,157.377
C05108=1047.117,262.308,395.555,171.896,38.891,157.377
C05109=1047.110,262.060,395.585,171.893,38.888,157.376
C05110=1047.103,261.811,395.614,171.891,38.886,157.375
C05111=1047.097,261.564,395.644,171.888,38.883,157.375
C05112=1047.090,261.315,395.673,171.884,38.880,157.374
C05113=1047.083,261.067,395.703,171.882,38.878,157.373
C05114=1047.076,260.819,395.733,171.879,38.875,157.373
C05115=1047.070,260.571,395.762,171.877,38.872,157.372
C05116=1047.063,260.322,395.792,171.874,38.870,157.371
C05117=1047.056,260.075,395.821,171.871,38.867,157.371
C05118=1047.050,259.826,395.851,171.868,38.864,157.370
C05119=1047.043,259.578,395.881,171.865,38.861,157.369
C05120=1047.036,259.330,395.910,171.863,38.859,157.369
C05121=1047.030,259.081,395.939,171.860,38.856,157.368
C05122=1047.023,258.834,395.969,171.857,38.853,157.367
C05123=1047.016,258.585,395.998,171.854,38.851,157.367
C05124=1047.010,258.338,396.028,171.851,38.848,157.366
C05125=1047.003,258.089,396.057,171.849,38.845,157.366
C05126=1046.997,257.841,396.086,171.846,38.842,157.365
C05127=1046.990,257.593,396.116,171.844,38.840,157.364
C05128=1046.983,257.344,396.146,171.841,38.837,157.364
C05129=1046.977,257.096,396.175,171.837,38.834,157.363
C05130=1046.970,256.848,396.203,171.835,38.832,157.362
C05131=1046.963,256.600,396.233,171.832,38.829,157.362
C05132=1046.957,256.352,396.262,171.830,38.826,157.361
C05133=1046.950,256.103,396.292,171.827,38.823,157.360
C05134=1046.944,255.855,396.321,171.825,38.821,157.360
C05135=1046.937,255.607,396.350,171.822,38.818,157.359
C05136=1046.930,255.359,396.380,171.819,38.815,157.358
C05137=1046.924,255.111,396.409,171.816,38.813,157.358
C05138=1046.918,254.862,396.438,171.813,38.810,157.357
C05139=1046.911,254.614,396.467,171.811,38.807,157.356
C05140=1046.904,254.366,396.497,171.808,38.805,157.356
C05141=1046.898,254.118,396.526,171.805,38.802,157.355
C05142=1046.892,253.870,396.555,171.803,38.799,157.354
C05143=1046.884,253.621,396.584,171.800,38.797,157.354
C05144=1046.878,253.373,396.613,171.798,38.794,157.353
C05145=1046.872,253.125,396.642,171.795,38.791,157.353
C05146=1046.866,252.877,396.671,171.792,38.788,157.352
C05147=1046.859,252.628,396.701,171.789,38.786,157.351
C05148=1046.852,252.381,396.730,171.786,38.783,157.351
C05149=1046.846,252.132,396.759,171.784,38.780,157.350
C05150=1046.840,251.884,396.788,171.781,38.778,157.349
C05151=1046.833,251.635,396.818,171.778,38.775,157.349
C05152=1046.827,251.387,396.847,171.776,38.772,157.348
C05153=1046.820,251.139,396.875,171.773,38.770,157.347
C05154=1046.813,250.891,396.904,171.771,38.767,157.347
C05155=1046.807,250.643,396.933,171.768,38.764,157.346
C05156=1046.800,250.394,396.963,171.766,38.761,157.345
C05157=1046.794,250.146,396.992,171.763,38.759,157.345
C05158=1046.788,249.898,397.021,171.760,38.756,157.344
C05159=1046.781,249.650,397.050,171.758,38.753,157.343
C05160=1046.775,249.402,397.079,171.755,38.750,157.343
C05161=1046.768,249.133,397.110,171.753,38.747,157.342
C05162=1046.761,248.865,397.141,171.750,38.744,157.341
C05163=1046.754,248.595,397.172,171.746,38.741,157.341
C05164=1046.747,248.326,397.204,171.744,38.738,157.340
C05165=1046.741,248.078,397.233,171.741,38.735,157.339
C05166=1046.735,247.830,397.262,171.739,38.733,157.339
C05167=1046.728,247.582,397.291,171.736,38.730,157.338
C05168=1046.721,247.334,397.319,171.733,38.727,157.337
C05169=1046.715,247.086,397.348,171.731,38.725,157.337
C05170=1046.709,246.838,397.377,171.728,38.722,157.336
C05171=1046.703,246.589,397.406,171.726,38.719,157.335
C05172=1046.696,246.340,397.435,171.723,38.716,157.335
C05173=1046.690,246.092,397.464,171.720,38.714,157.334
C05174=1046.684,245.844,397.493,171.718,38.711,157.333
C05175=1046.677,245.596,397.521,171.715,38.708,157.333
C05176=1046.671,245.347,397.550,171.713,38.705,157.332
C05177=1046.664,245.099,397.579,171.710,38.703,157.331
C05178=1046.657,244.852,397.607,171.708,38.700,157.331
C05179=1046.651,244.603,397.636,171.705,38.697,157.330
C05180=1046.645,244.355,397.665,171.702,38.694,157.330
C05181=1046.639,244.106,397.692,171.700,38.692,157.329
C05182=1046.632,243.858,397.721,171.698,38.689,157.328
C05183=1046.625,243.610,397.750,171.696,38.686,157.328
C05184=1046.619,243.361,397.779,171.693,38.683,157.327
C05185=1046.613,243.113,397.808,171.691,38.681,157.326
C05186=1046.606,242.865,397.836,171.688,38.678,157.326
C05187=1046.600,242.616,397.864,171.685,38.675,157.325
C05188=1046.593,242.368,397.893,171.683,38.672,157.324
C05189=1046.587,242.120,397.921,171.680,38.670,157.324
C05190=1046.580,241.871,397.950,171.678,38.667,157.323
C05191=1046.574,241.623,397.978,171.675,38.664,157.322
C05192=1046.567,241.375,398.007,171.673,38.661,157.322
C05193=1046.561,241.126,398.035,171.670,38.659,157.321
C05194=1046.554,240.879,398.063,171.668,38.656,157.321
C05195=1046.548,240.630,398.092,171.665,38.654,157.320
C05196=1046.541,240.382,398.120,171.662,38.651,157.319
C05197=1046.535,240.133,398.148,171.660,38.648,157.319
C05198=1046.528,239.885,398.176,171.657,38.646,157.318
C05199=1046.521,239.637,398.204,171.656,38.643,157.317
C05200=1046.515,239.388,398.233,171.653,38.641,157.317
C05201=1046.508,239.140,398.261,171.651,38.638,157.316
C05202=1046.502,238.892,398.289,171.648,38.635,157.316
C05203=1046.496,238.643,398.317,171.646,38.632,157.315
C05204=1046.489,238.395,398.346,171.643,38.630,157.314
C05205=1046.482,238.147,398.373,171.640,38.627,157.314
C05206=1046.476,237.898,398.402,171.638,38.624,157.313
C05207=1046.469,237.650,398.430,171.635,38.621,157.312
C05208=1046.462,237.402,398.458,171.633,38.618,157.312
C05209=1046.456,237.153,398.486,171.630,38.616,157.311
C05210=1046.450,236.905,398.514,171.629,38.613,157.311
C05211=1046.443,236.657,398.542,171.626,38.611,157.310
C05212=1046.436,236.408,398.570,171.624,38.608,157.309
C05213=1046.430,236.160,398.599,171.621,38.605,157.309
C05214=1046.424,235.911,398.626,171.618,38.603,157.308
C05215=1046.417,235.663,398.654,171.616,38.600,157.307
C05216=1046.411,235.415,398.683,171.613,38.597,157.307
C05217=1046.403,235.140,398.713,171.611,38.594,157.306
C05218=1046.396,234.866,398.744,171.608,38.591,157.305
C05219=1046.389,234.591,398.775,171.606,38.588,157.305
C05220=1046.382,234.317,398.806,171.603,38.585,157.304
C05221=1046.375,234.068,398.834,171.600,38.582,157.303
C05222=1046.369,233.820,398.862,171.598,38.580,157.303
C05223=1046.363,233.572,398.889,171.596,38.577,157.302
C05224=1046.357,233.323,398.918,171.594,38.574,157.301
C05225=1046.350,233.075,398.946,171.591,38.571,157.301
C05226=1046.343,232.827,398.974,171.589,38.569,157.300
C05227=1046.336,232.578,399.001,171.586,38.566,157.300
C05228=1046.330,232.330,399.030,171.583,38.563,157.299
C05229=1046.324,232.081,399.058,171.582,38.561,157.298
C05230=1046.317,231.833,399.085,171.579,38.558,157.298
C05231=1046.311,231.585,399.113,171.577,38.556,157.297
C05232=1046.304,231.337,399.140,171.574,38.553,157.296
C05233=1046.298,231.088,399.168,171.572,38.550,157.296
C05234=1046.291,230.840,399.196,171.570,38.547,157.295
C05235=1046.284,230.591,399.224,171.568,38.544,157.295
C05236=1046.278,230.343,399.252,171.565,38.542,157.294
C05237=1046.272,230.094,399.280,171.563,38.539,157.293
C05238=1046.265,229.846,399.307,171.560,38.536,157.293
C05239=1046.259,229.598,399.335,171.557,38.533,157.292
C05240=1046.252,229.349,399.362,171.556,38.531,157.292
C05241=1046.246,229.100,399.389,171.553,38.528,157.291
C05242=1046.239,228.852,399.417,171.551,38.525,157.290
C05243=1046.233,228.604,399.445,171.548,38.523,157.290
C05244=1046.226,228.356,399.472,171.547,38.520,157.289
C05245=1046.220,228.107,399.500,171.544,38.518,157.288
C05246=1046.213,227.858,399.527,171.542,38.515,157.288
C05247=1046.207,227.610,399.555,171.539,38.512,157.287
C05248=1046.200,227.361,399.582,171.537,38.509,157.287
C05249=1046.194,227.114,399.610,171.535,38.506,157.286
C05250=1046.186,226.866,399.637,171.533,38.504,157.285
C05251=1046.180,226.617,399.664,171.530,38.501,157.285
C05252=1046.173,226.368,399.692,171.528,38.499,157.284
C05253=1046.167,226.120,399.719,171.526,38.496,157.283
C05254=1046.161,225.871,399.746,171.523,38.493,157.283
C05255=1046.154,225.623,399.774,171.521,38.491,157.282
C05256=1046.147,225.374,399.802,171.518,38.488,157.282
C05257=1046.141,225.126,399.829,171.516,38.485,157.281
C05258=1046.135,224.878,399.856,171.514,38.482,157.280
C05259=1046.128,224.629,399.883,171.512,38.479,157.280
C05260=1046.121,224.381,399.911,171.509,38.477,157.279
C05261=1046.115,224.132,399.938,171.508,38.474,157.278
C05262=1046.108,223.884,399.965,171.505,38.471,157.278
C05263=1046.102,223.636,399.993,171.503,38.469,157.277
C05264=1046.095,223.387,400.020,171.500,38.466,157.277
C05265=1046.089,223.138,400.048,171.498,38.463,157.276
C05266=1046.082,222.890,400.074,171.496,38.461,157.275
C05267=1046.076,222.642,400.101,171.493,38.458,157.275
C05268=1046.069,222.393,400.128,171.491,38.455,157.274
C05269=1046.063,222.145,400.156,171.489,38.452,157.274
C05270=1046.056,221.897,400.184,171.487,38.450,157.273
C05271=1046.050,221.647,400.211,171.484,38.447,157.272
C05272=1046.044,221.400,400.238,171.483,38.444,157.272
C05273=1046.036,221.117,400.269,171.480,38.441,157.271
C05274=1046.028,220.836,400.299,171.478,38.438,157.270
C05275=1046.021,220.554,400.330,171.475,38.435,157.270
C05276=1046.014,220.271,400.361,171.472,38.432,157.269
C05277=1046.007,220.023,400.388,171.470,38.429,157.268
C05278=1046.001,219.775,400.415,171.468,38.426,157.268
C05279=1045.994,219.526,400.441,171.466,38.424,157.267
C05280=1045.988,219.277,400.469,171.463,38.421,157.266
C05281=1045.981,219.029,400.495,171.462,38.418,157.266
C05282=1045.974,218.781,400.523,171.459,38.415,157.265
C05283=1045.968,218.532,400.550,171.457,38.413,157.264
C05284=1045.962,218.284,400.576,171.454,38.410,157.264
C05285=1045.955,218.035,400.604,171.453,38.407,157.263
C05286=1045.948,217.787,400.630,171.450,38.405,157.263
C05287=1045.942,217.538,400.657,171.448,38.402,157.262
C05288=1045.935,217.290,400.684,171.446,38.399,157.261
C05289=1045.928,217.041,400.711,171.443,38.397,157.261
C05290=1045.922,216.793,400.738,171.441,38.394,157.260
C05291=1045.915,216.545,400.765,171.439,38.391,157.260
C05292=1045.909,216.296,400.791,171.437,38.388,157.259
C05293=1045.902,216.048,400.818,171.435,38.385,157.258
C05294=1045.896,215.798,400.845,171.433,38.383,157.258
C05295=1045.890,215.551,400.872,171.430,38.380,157.257
C05296=1045.883,215.302,400.899,171.429,38.377,157.256
C05297=1045.877,215.054,400.925,171.426,38.375,157.256
C05298=1045.870,214.805,400.952,171.424,38.372,157.255
C05299=1045.864,214.557,400.979,171.422,38.369,157.255
C05300=1045.856,214.308,401.005,171.420,38.367,157.254
C05301=1045.850,214.059,401.032,171.418,38.364,157.253
C05302=1045.844,213.811,401.058,171.416,38.361,157.253
C05303=1045.837,213.562,401.085,171.413,38.358,157.252
C05304=1045.831,213.314,401.112,171.412,38.355,157.252
C05305=1045.824,213.066,401.139,171.409,38.352,157.251
C05306=1045.818,212.817,401.166,171.407,38.349,157.250
C05307=1045.811,212.569,401.192,171.405,38.347,157.250
C05308=1045.805,212.320,401.219,171.402,38.344,157.249
C05309=1045.798,212.072,401.245,171.401,38.341,157.248
C05310=1045.792,211.823,401.272,171.398,38.339,157.248
C05311=1045.785,211.574,401.298,171.397,38.336,157.247
C05312=1045.780,211.326,401.325,171.394,38.333,157.247
C05313=1045.772,211.077,401.352,171.392,38.330,157.246
C05314=1045.766,210.829,401.378,171.390,38.327,157.245
C05315=1045.760,210.580,401.405,171.388,38.325,157.245
C05316=1045.752,210.331,401.431,171.386,38.322,157.244
C05317=1045.747,210.083,401.458,171.384,38.319,157.243
C05318=1045.740,209.835,401.484,171.381,38.316,157.243
C05319=1045.733,209.586,401.510,171.380,38.314,157.242
C05320=1045.727,209.338,401.537,171.377,38.311,157.242
C05321=1045.720,209.089,401.563,171.376,38.308,157.241
C05322=1045.714,208.841,401.589,171.373,38.306,157.240
C05323=1045.707,208.592,401.616,171.372,38.303,157.240
C05324=1045.701,208.344,401.642,171.369,38.300,157.239
C05325=1045.694,208.095,401.669,171.368,38.297,157.239
C05326=1045.687,207.847,401.695,171.365,38.294,157.238
C05327=1045.681,207.598,401.722,171.362,38.291,157.237
C05328=1045.674,207.350,401.748,171.361,38.288,157.237
C05329=1045.667,207.073,401.776,171.358,38.285,157.236
C05330=1045.660,206.797,401.806,171.356,38.282,157.235
C05331=1045.652,206.520,401.836,171.354,38.279,157.235
C05332=1045.645,206.243,401.864,171.352,38.277,157.234
C05333=1045.619,205.192,401.971,171.096,38.176,157.208
C05334=1045.613,204.943,401.996,171.093,38.174,157.208
C05335=1045.607,204.694,402.021,171.090,38.172,157.207
C05336=1045.601,204.446,402.046,171.088,38.170,157.207
C05337=1045.595,204.198,402.071,171.085,38.168,157.206
C05338=1045.588,203.949,402.097,171.082,38.166,157.206
C05339=1045.583,203.700,402.121,171.080,38.164,157.206
C05340=1045.576,203.451,402.147,171.076,38.162,157.205
C05341=1045.569,203.203,402.172,171.074,38.160,157.205
C05342=1045.564,202.955,402.197,171.071,38.158,157.204
C05343=1045.558,202.706,402.221,171.068,38.156,157.204
C05344=1045.552,202.457,402.246,171.066,38.154,157.203
C05345=1045.546,202.208,402.272,171.063,38.152,157.203
C05346=1045.540,201.959,402.296,171.060,38.150,157.202
C05347=1045.534,201.711,402.321,171.058,38.148,157.202
C05348=1045.528,201.462,402.347,171.055,38.146,157.202
C05349=1045.522,201.213,402.371,171.052,38.144,157.201
C05350=1045.515,200.965,402.396,171.049,38.142,157.201
C05351=1045.509,200.716,402.421,171.046,38.140,157.200
C05352=1045.503,200.467,402.446,171.044,38.139,157.200
C05353=1045.497,200.219,402.470,171.041,38.137,157.199
C05354=1045.491,199.970,402.495,171.038,38.135,157.199
C05355=1045.484,199.721,402.520,171.036,38.133,157.198
C05356=1045.478,199.472,402.544,171.033,38.131,157.198
C05357=1045.471,199.224,402.569,171.030,38.129,157.198
C05358=1045.466,198.975,402.593,171.028,38.128,157.197
C05359=1045.459,198.726,402.619,171.025,38.126,157.197
C05360=1045.453,198.478,402.643,171.022,38.124,157.196
C05361=1045.446,198.229,402.668,171.020,38.122,157.196
C05362=1045.440,197.981,402.692,171.016,38.120,157.195
C05363=1045.434,197.732,402.717,171.014,38.118,157.195
C05364=1045.428,197.483,402.742,171.012,38.117,157.195
C05365=1045.422,197.234,402.766,171.008,38.115,157.194
C05366=1045.416,196.986,402.791,171.006,38.113,157.194
C05367=1045.409,196.737,402.815,171.004,38.111,157.193
C05368=1045.403,196.488,402.840,171.000,38.109,157.193
C05369=1045.397,196.239,402.864,170.998,38.107,157.193
C05370=1045.391,195.990,402.888,170.996,38.105,157.192
C05371=1045.385,195.742,402.914,170.993,38.104,157.192
C05372=1045.378,195.493,402.938,170.990,38.102,157.191
C05373=1045.373,195.244,402.962,170.987,38.100,157.191
C05374=1045.366,194.996,402.987,170.985,38.098,157.190
C05375=1045.360,194.747,403.011,170.982,38.096,157.190
C05376=1045.354,194.498,403.035,170.980,38.094,157.190
C05377=1045.348,194.250,403.060,170.977,38.093,157.189
C05378=1045.341,194.001,403.084,170.974,38.091,157.189
C05379=1045.336,193.752,403.109,170.972,38.089,157.188
C05380=1045.330,193.503,403.134,170.969,38.087,157.188
C05381=1045.323,193.254,403.158,170.967,38.085,157.187
C05382=1045.318,193.006,403.182,170.963,38.083,157.187
C05383=1045.311,192.757,403.206,170.961,38.082,157.187
C05384=1045.306,192.508,403.231,170.959,38.080,157.186
C05385=1045.299,192.260,403.255,170.955,38.078,157.186
C05386=1045.293,192.011,403.280,170.953,38.076,157.185
C05387=1045.287,191.762,403.304,170.951,38.075,157.185
C05388=1045.281,191.513,403.328,170.949,38.073,157.185
C05389=1045.275,191.265,403.352,170.945,38.071,157.184
C05390=1045.269,191.016,403.377,170.943,38.069,157.184
C05391=1045.263,190.768,403.401,170.941,38.068,157.183
C05392=1045.257,190.519,403.426,170.938,38.065,157.183
C05393=1045.250,190.270,403.450,170.935,38.063,157.183
C05394=1045.245,189.985,403.477,170.932,38.062,157.182
C05395=1045.237,189.701,403.505,170.929,38.059,157.182
C05396=1045.230,189.416,403.533,170.927,38.058,157.181
C05397=1045.223,189.132,403.561,170.923,38.055,157.181
C05398=1045.218,188.883,403.585,170.921,38.053,157.180
C05399=1045.211,188.634,403.609,170.919,38.052,157.180
C05400=1045.206,188.386,403.633,170.915,38.050,157.180
C05401=1045.199,188.137,403.657,170.913,38.048,157.179
C05402=1045.194,187.888,403.681,170.911,38.046,157.179
C05403=1045.187,187.639,403.705,170.908,38.045,157.178
C05404=1045.182,187.391,403.730,170.906,38.043,157.178
C05405=1045.176,187.142,403.753,170.903,38.041,157.178
C05406=1045.170,186.893,403.778,170.900,38.039,157.177
C05407=1045.164,186.645,403.802,170.898,38.038,157.177
C05408=1045.158,186.395,403.826,170.896,38.036,157.176
C05409=1045.152,186.147,403.850,170.893,38.034,157.176
C05410=1045.146,185.898,403.875,170.890,38.032,157.176
C05411=1045.140,185.650,403.898,170.888,38.031,157.175
C05412=1045.134,185.400,403.923,170.885,38.029,157.175
C05413=1045.128,185.152,403.947,170.883,38.027,157.174
C05414=1045.123,184.903,403.971,170.881,38.025,157.174
C05415=1045.116,184.654,403.994,170.877,38.023,157.173
C05416=1045.110,184.406,404.018,170.875,38.021,157.173
C05417=1045.105,184.156,404.042,170.873,38.019,157.173
C05418=1045.098,183.908,404.066,170.870,38.018,157.172
C05419=1045.093,183.659,404.091,170.868,38.017,157.172
C05420=1045.087,183.410,404.114,170.865,38.015,157.172
C05421=1045.079,183.161,404.137,170.863,38.013,157.171
C05422=1045.073,182.913,404.161,170.860,38.011,157.171
C05423=1045.067,182.664,404.185,170.858,38.010,157.171
C05424=1045.061,182.415,404.208,170.856,38.008,157.170
C05425=1045.054,182.166,404.232,170.852,38.007,157.170
C05426=1045.048,181.918,404.255,170.850,38.005,157.169
C05427=1045.042,181.668,404.279,170.848,38.004,157.169
C05428=1045.036,181.420,404.302,170.846,38.002,157.169
C05429=1045.029,181.171,404.326,170.843,38.000,157.168
C05430=1045.024,180.922,404.349,170.840,37.999,157.168
C05431=1045.018,180.674,404.373,170.838,37.997,157.168
C05432=1045.011,180.424,404.396,170.835,37.996,157.167
C05433=1045.005,180.176,404.420,170.833,37.994,157.167
C05434=1044.999,179.927,404.444,170.831,37.993,157.167
C05435=1044.993,179.678,404.467,170.828,37.991,157.166
C05436=1044.986,179.429,404.490,170.825,37.989,157.166
C05437=1044.980,179.180,404.513,170.823,37.988,157.165
C05438=1044.974,178.932,404.537,170.821,37.986,157.165
C05439=1044.967,178.682,404.560,170.818,37.984,157.165
C05440=1044.961,178.434,404.584,170.815,37.983,157.164
C05441=1044.955,178.185,404.607,170.813,37.982,157.164
C05442=1044.949,177.936,404.631,170.811,37.980,157.164
C05443=1044.943,177.687,404.654,170.808,37.979,157.163
C05444=1044.937,177.438,404.678,170.806,37.977,157.163
C05445=1044.931,177.190,404.701,170.804,37.975,157.163
C05446=1044.925,176.941,404.724,170.802,37.974,157.162
C05447=1044.918,176.692,404.747,170.798,37.972,157.162
C05448=1044.912,176.444,404.771,170.796,37.970,157.161
C05449=1044.905,176.194,404.794,170.794,37.969,157.161
C05450=1044.899,175.946,404.818,170.791,37.967,157.161
C05451=1044.894,175.697,404.841,170.789,37.966,157.160
C05452=1044.887,175.447,404.864,170.787,37.965,157.160
C05453=1044.881,175.199,404.888,170.784,37.963,157.160
C05454=1044.876,174.950,404.911,170.781,37.961,157.159
C05455=1044.869,174.702,404.934,170.779,37.960,157.159
C05456=1044.862,174.453,404.957,170.777,37.958,157.159
C05457=1044.857,174.204,404.980,170.774,37.956,157.158
C05458=1044.850,173.919,405.007,170.772,37.955,157.158
